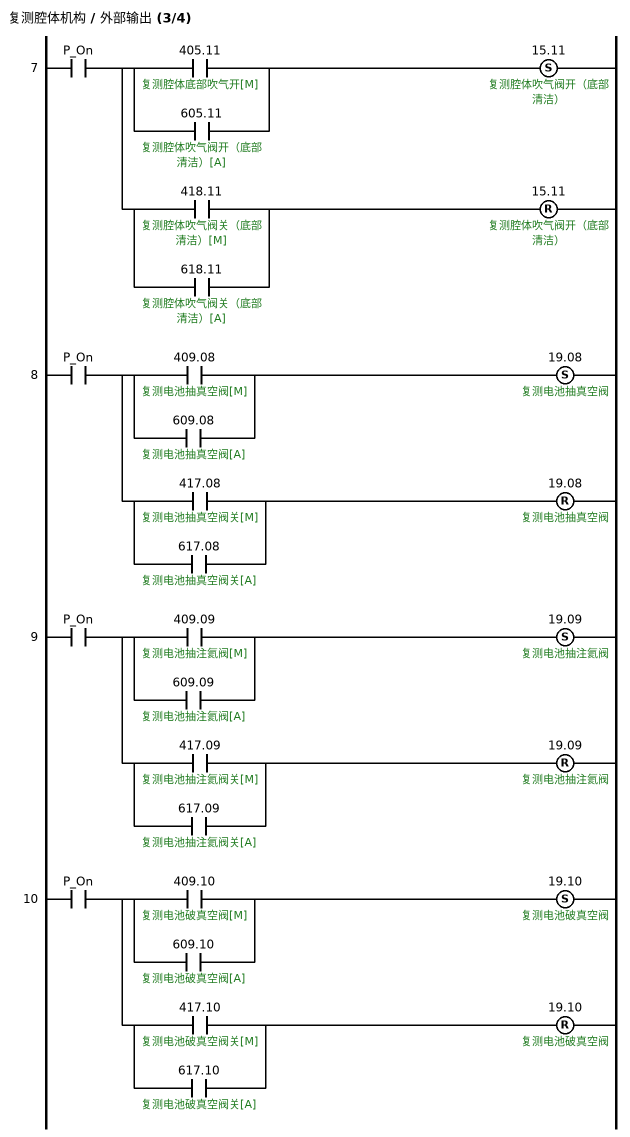
; [picture p624: 复测腔体机构 / 外部输出, rungs 7-10]
; rung 7
LD P_On
OUT TR0
LD 405.11  ; 复测腔体底部吹气开[M]
OR 605.11  ; 复测腔体吹气阀开（底部清洁）[A]
ANDLD
SET 15.11  ; 复测腔体吹气阀开（底部清洁）
LD TR0
LD 418.11  ; 复测腔体吹气阀关（底部清洁）[M]
OR 618.11  ; 复测腔体吹气阀关（底部清洁）[A]
ANDLD
RSET 15.11  ; 复测腔体吹气阀开（底部清洁）
; rung 8
LD P_On
OUT TR0
LD 409.08  ; 复测电池抽真空阀[M]
OR 609.08  ; 复测电池抽真空阀[A]
ANDLD
SET 19.08  ; 复测电池抽真空阀
LD TR0
LD 417.08  ; 复测电池抽真空阀关[M]
OR 617.08  ; 复测电池抽真空阀关[A]
ANDLD
RSET 19.08  ; 复测电池抽真空阀
; rung 9
LD P_On
OUT TR0
LD 409.09  ; 复测电池抽注氦阀[M]
OR 609.09  ; 复测电池抽注氦阀[A]
ANDLD
SET 19.09  ; 复测电池抽注氦阀
LD TR0
LD 417.09  ; 复测电池抽注氦阀关[M]
OR 617.09  ; 复测电池抽注氦阀关[A]
ANDLD
RSET 19.09  ; 复测电池抽注氦阀
; rung 10
LD P_On
OUT TR0
LD 409.10  ; 复测电池破真空阀[M]
OR 609.10  ; 复测电池破真空阀[A]
ANDLD
SET 19.10  ; 复测电池破真空阀
LD TR0
LD 417.10  ; 复测电池破真空阀关[M]
OR 617.10  ; 复测电池破真空阀关[A]
ANDLD
RSET 19.10  ; 复测电池破真空阀

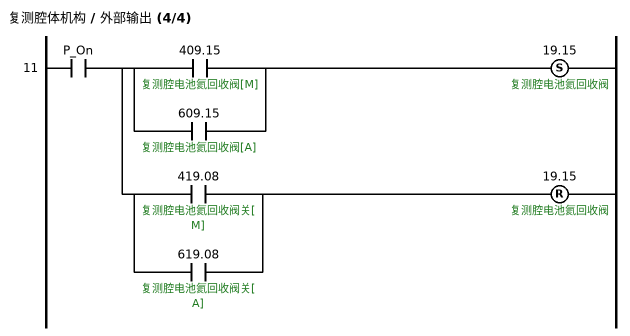
; rung 11
LD P_On
OUT TR0
LD 409.15  ; 复测腔电池氦回收阀[M]
OR 609.15  ; 复测腔电池氦回收阀[A]
ANDLD
SET 19.15  ; 复测腔电池氦回收阀
LD TR0
LD 419.08  ; 复测腔电池氦回收阀关[M]
OR 619.08  ; 复测腔电池氦回收阀关[A]
ANDLD
RSET 19.15  ; 复测腔电池氦回收阀

### Section END
; rung 0
END(001)

## Program Common (cyclic task 8)

### Section 动作延时

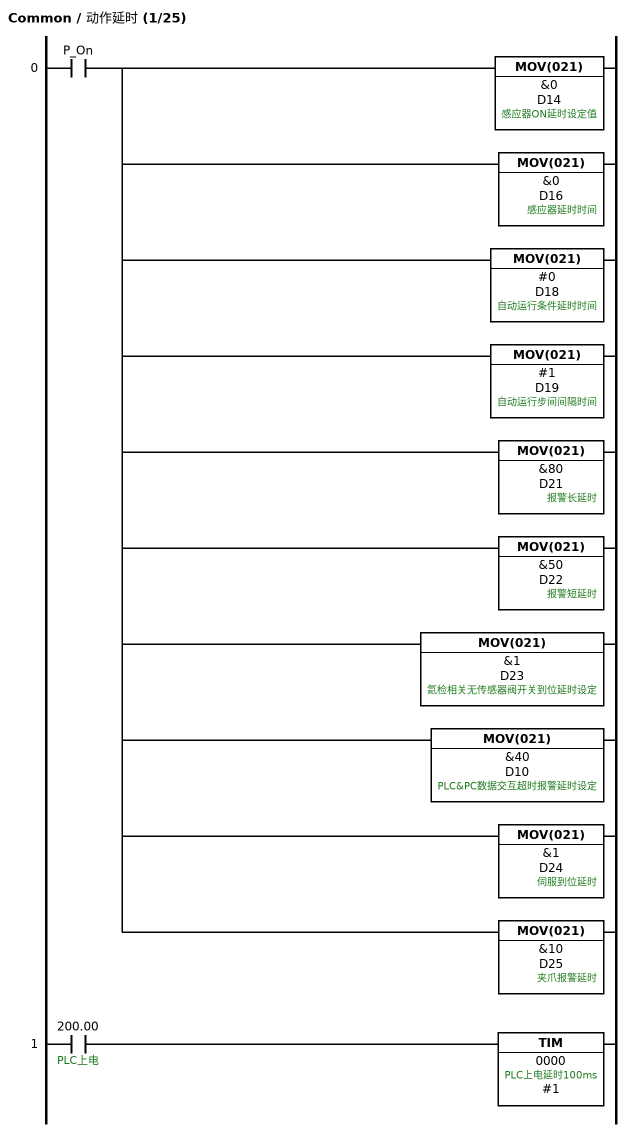
; rung 0
LD P_On
MOV(021) &0 D14  ; 感应器ON延时设定值
MOV(021) &0 D16  ; 感应器延时时间
MOV(021) #0 D18  ; 自动运行条件延时时间
MOV(021) #1 D19  ; 自动运行步间间隔时间
MOV(021) &80 D21  ; 报警长延时
MOV(021) &50 D22  ; 报警短延时
MOV(021) &1 D23  ; 氦检相关无传感器阀开关到位延时设定
MOV(021) &40 D10  ; PLC&PC数据交互超时报警延时设定
MOV(021) &1 D24  ; 伺服到位延时
MOV(021) &10 D25  ; 夹爪报警延时
; rung 1
LD 200.00  ; PLC上电
TIM 0000 #1  ; PLC上电延时100ms

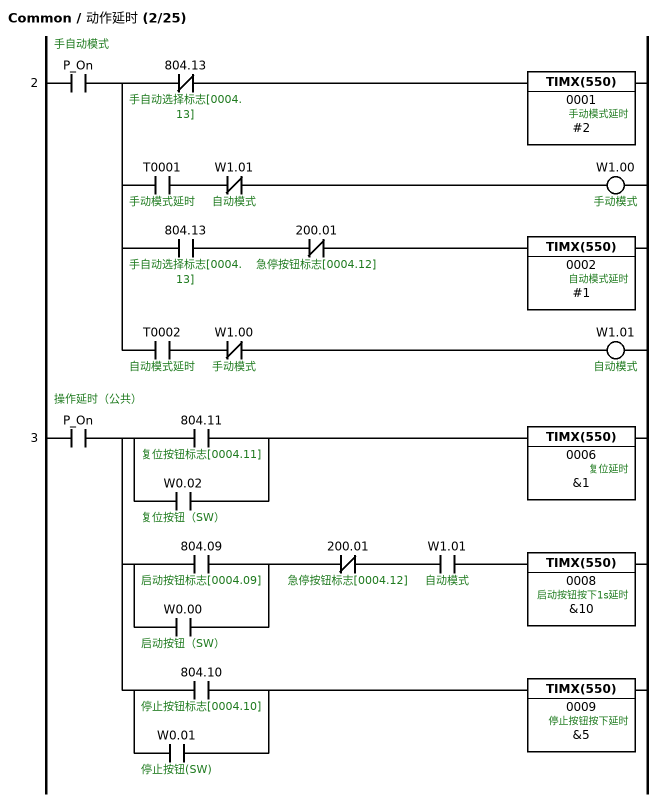
; rung 2: 手自动模式
LD P_On
OUT TR0
ANDNOT 804.13  ; 手自动选择标志[0004.13]
TIMX(550) 0001 #2  ; 手动模式延时
LD TR0
AND T0001  ; 手动模式延时
ANDNOT W1.01  ; 自动模式
OUT W1.00  ; 手动模式
LD TR0
AND 804.13  ; 手自动选择标志[0004.13]
ANDNOT 200.01  ; 急停按钮标志[0004.12]
TIMX(550) 0002 #1  ; 自动模式延时
LD TR0
AND T0002  ; 自动模式延时
ANDNOT W1.00  ; 手动模式
OUT W1.01  ; 自动模式
; rung 3: 操作延时（公共）
LD P_On
OUT TR0
LD 804.11  ; 复位按钮标志[0004.11]
OR W0.02  ; 复位按钮（SW）
ANDLD
TIMX(550) 0006 &1  ; 复位延时
LD TR0
LD 804.09  ; 启动按钮标志[0004.09]
OR W0.00  ; 启动按钮（SW）
ANDLD
ANDNOT 200.01  ; 急停按钮标志[0004.12]
AND W1.01  ; 自动模式
TIMX(550) 0008 &10  ; 启动按钮按下1s延时
LD TR0
LD 804.10  ; 停止按钮标志[0004.10]
OR W0.01  ; 停止按钮(SW)
ANDLD
TIMX(550) 0009 &5  ; 停止按钮按下延时

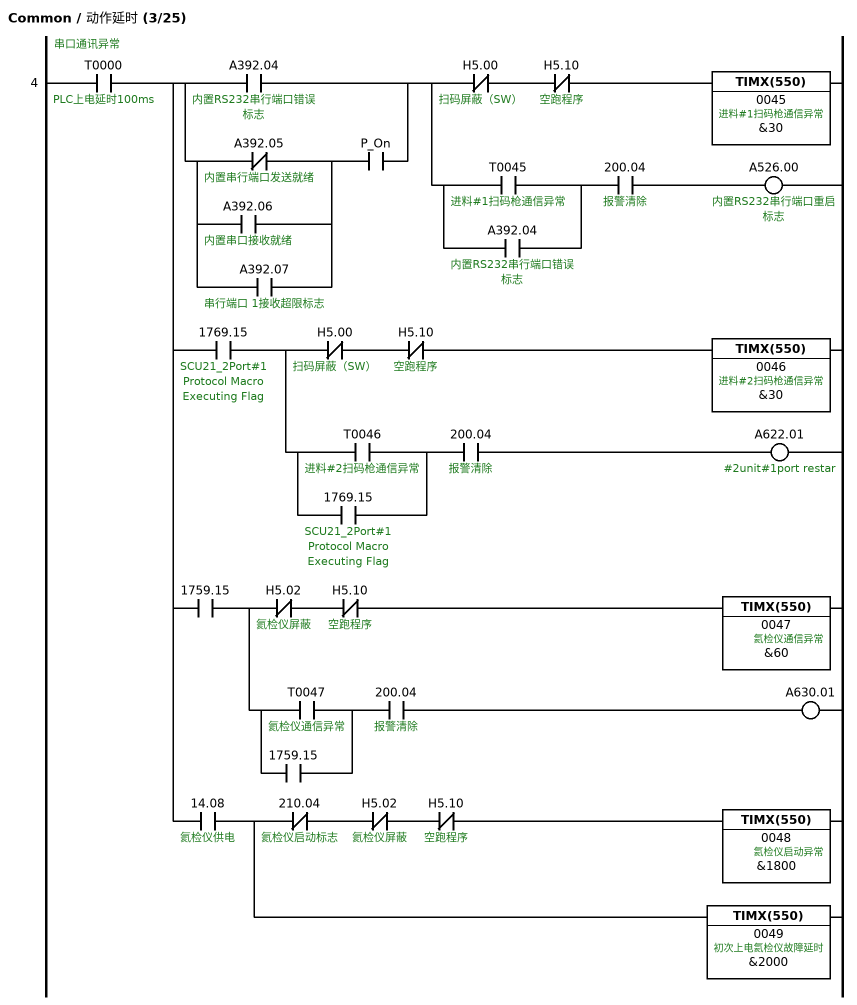
; rung 4: 串口通讯异常
LD T0000  ; PLC上电延时100ms
OUT TR0
LD A392.04  ; 内置RS232串行端口错误标志
LDNOT A392.05  ; 内置串行端口发送就绪
OR A392.06  ; 内置串口接收就绪
OR A392.07  ; 串行端口 1接收超限标志
AND P_On
ORLD
ANDLD
OUT TR1
ANDNOT H5.00  ; 扫码屏蔽（SW）
ANDNOT H5.10  ; 空跑程序
TIMX(550) 0045 &30  ; 进料#1扫码枪通信异常
LD TR1
LD T0045  ; 进料#1扫码枪通信异常
OR A392.04  ; 内置RS232串行端口错误标志
ANDLD
AND 200.04  ; 报警清除
OUT A526.00  ; 内置RS232串行端口重启标志
LD TR0
AND 1769.15  ; SCU21_2Port#1 Protocol Macro Executing Flag
OUT TR1
ANDNOT H5.00  ; 扫码屏蔽（SW）
ANDNOT H5.10  ; 空跑程序
TIMX(550) 0046 &30  ; 进料#2扫码枪通信异常
LD TR1
LD T0046  ; 进料#2扫码枪通信异常
OR 1769.15  ; SCU21_2Port#1 Protocol Macro Executing Flag
ANDLD
AND 200.04  ; 报警清除
OUT A622.01  ; #2unit#1port restar
LD TR0
AND 1759.15
OUT TR1
ANDNOT H5.02  ; 氦检仪屏蔽
ANDNOT H5.10  ; 空跑程序
TIMX(550) 0047 &60  ; 氦检仪通信异常
LD TR1
LD T0047  ; 氦检仪通信异常
OR 1759.15
ANDLD
AND 200.04  ; 报警清除
OUT A630.01
LD TR0
AND 14.08  ; 氦检仪供电
OUT TR0
ANDNOT 210.04  ; 氦检仪启动标志
ANDNOT H5.02  ; 氦检仪屏蔽
ANDNOT H5.10  ; 空跑程序
TIMX(550) 0048 &1800  ; 氦检仪启动异常
LD TR0
TIMX(550) 0049 &2000  ; 初次上电氦检仪故障延时

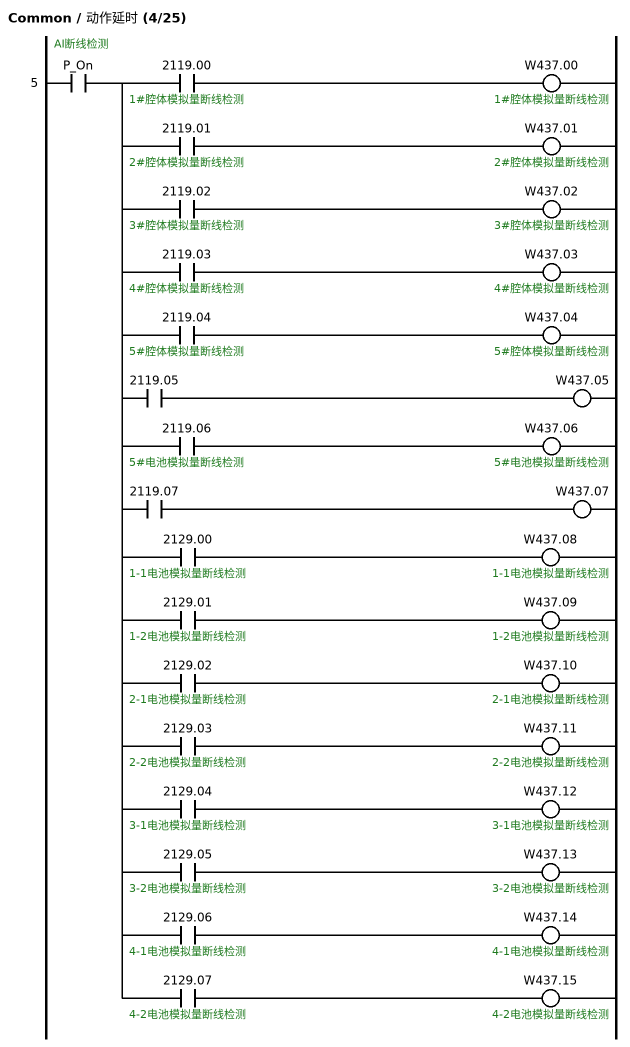
; rung 5: AI断线检测
LD P_On
OUT TR0
AND 2119.00  ; 1#腔体模拟量断线检测
OUT W437.00  ; 1#腔体模拟量断线检测
LD TR0
AND 2119.01  ; 2#腔体模拟量断线检测
OUT W437.01  ; 2#腔体模拟量断线检测
LD TR0
AND 2119.02  ; 3#腔体模拟量断线检测
OUT W437.02  ; 3#腔体模拟量断线检测
LD TR0
AND 2119.03  ; 4#腔体模拟量断线检测
OUT W437.03  ; 4#腔体模拟量断线检测
LD TR0
AND 2119.04  ; 5#腔体模拟量断线检测
OUT W437.04  ; 5#腔体模拟量断线检测
LD TR0
AND 2119.05
OUT W437.05
LD TR0
AND 2119.06  ; 5#电池模拟量断线检测
OUT W437.06  ; 5#电池模拟量断线检测
LD TR0
AND 2119.07
OUT W437.07
LD TR0
AND 2129.00  ; 1-1电池模拟量断线检测
OUT W437.08  ; 1-1电池模拟量断线检测
LD TR0
AND 2129.01  ; 1-2电池模拟量断线检测
OUT W437.09  ; 1-2电池模拟量断线检测
LD TR0
AND 2129.02  ; 2-1电池模拟量断线检测
OUT W437.10  ; 2-1电池模拟量断线检测
LD TR0
AND 2129.03  ; 2-2电池模拟量断线检测
OUT W437.11  ; 2-2电池模拟量断线检测
LD TR0
AND 2129.04  ; 3-1电池模拟量断线检测
OUT W437.12  ; 3-1电池模拟量断线检测
LD TR0
AND 2129.05  ; 3-2电池模拟量断线检测
OUT W437.13  ; 3-2电池模拟量断线检测
LD TR0
AND 2129.06  ; 4-1电池模拟量断线检测
OUT W437.14  ; 4-1电池模拟量断线检测
LD TR0
AND 2129.07  ; 4-2电池模拟量断线检测
OUT W437.15  ; 4-2电池模拟量断线检测

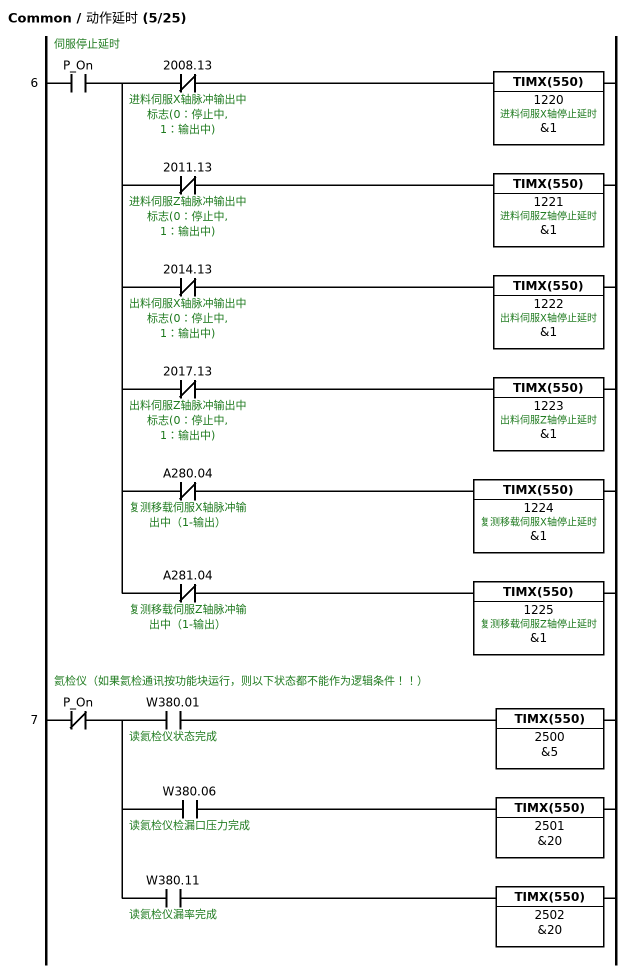
; rung 6: 伺服停止延时
LD P_On
OUT TR0
ANDNOT 2008.13  ; 进料伺服X轴脉冲输出中标志(0：停止中,1：输出中)
TIMX(550) 1220 &1  ; 进料伺服X轴停止延时
LD TR0
ANDNOT 2011.13  ; 进料伺服Z轴脉冲输出中标志(0：停止中,1：输出中)
TIMX(550) 1221 &1  ; 进料伺服Z轴停止延时
LD TR0
ANDNOT 2014.13  ; 出料伺服X轴脉冲输出中标志(0：停止中,1：输出中)
TIMX(550) 1222 &1  ; 出料伺服X轴停止延时
LD TR0
ANDNOT 2017.13  ; 出料伺服Z轴脉冲输出中标志(0：停止中,1：输出中)
TIMX(550) 1223 &1  ; 出料伺服Z轴停止延时
LD TR0
ANDNOT A280.04  ; 复测移载伺服X轴脉冲输出中（1-输出）
TIMX(550) 1224 &1  ; 复测移载伺服X轴停止延时
LD TR0
ANDNOT A281.04  ; 复测移载伺服Z轴脉冲输出中（1-输出）
TIMX(550) 1225 &1  ; 复测移载伺服Z轴停止延时
; rung 7: 氦检仪（如果氦检通讯按功能块运行，则以下状态都不能作为逻辑条件！！）
LDNOT P_On
OUT TR0
AND W380.01  ; 读氦检仪状态完成
TIMX(550) 2500 &5
LD TR0
AND W380.06  ; 读氦检仪检漏口压力完成
TIMX(550) 2501 &20
LD TR0
AND W380.11  ; 读氦检仪漏率完成
TIMX(550) 2502 &20

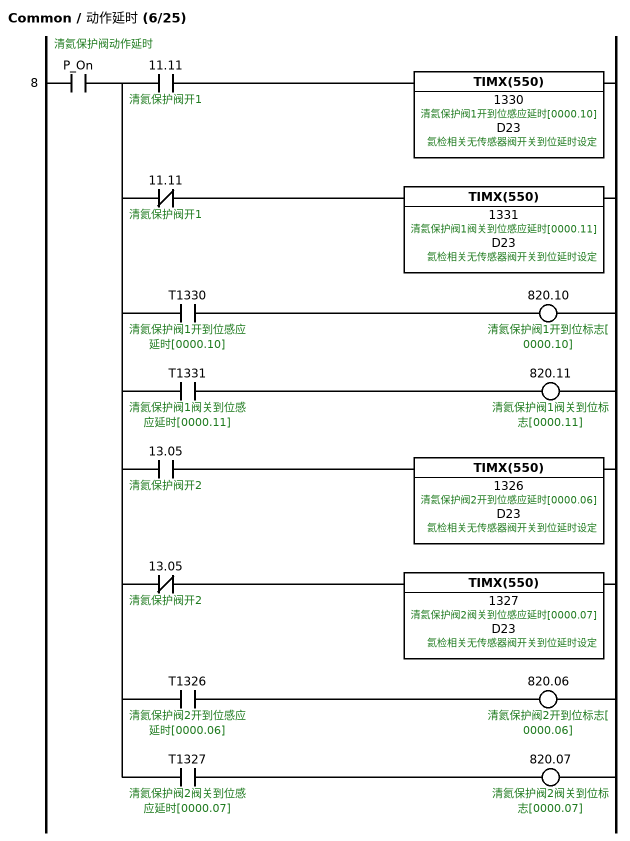
; rung 8: 清氦保护阀动作延时
LD P_On
OUT TR0
AND 11.11  ; 清氦保护阀开1
TIMX(550) 1330 D23  ; 氦检相关无传感器阀开关到位延时设定, 清氦保护阀1开到位感应延时[0000.10]
LD TR0
ANDNOT 11.11  ; 清氦保护阀开1
TIMX(550) 1331 D23  ; 氦检相关无传感器阀开关到位延时设定, 清氦保护阀1阀关到位感应延时[0000.11]
LD TR0
AND T1330  ; 清氦保护阀1开到位感应延时[0000.10]
OUT 820.10  ; 清氦保护阀1开到位标志[0000.10]
LD TR0
AND T1331  ; 清氦保护阀1阀关到位感应延时[0000.11]
OUT 820.11  ; 清氦保护阀1阀关到位标志[0000.11]
LD TR0
AND 13.05  ; 清氦保护阀开2
TIMX(550) 1326 D23  ; 氦检相关无传感器阀开关到位延时设定, 清氦保护阀2开到位感应延时[0000.06]
LD TR0
ANDNOT 13.05  ; 清氦保护阀开2
TIMX(550) 1327 D23  ; 氦检相关无传感器阀开关到位延时设定, 清氦保护阀2阀关到位感应延时[0000.07]
LD TR0
AND T1326  ; 清氦保护阀2开到位感应延时[0000.06]
OUT 820.06  ; 清氦保护阀2开到位标志[0000.06]
LD TR0
AND T1327  ; 清氦保护阀2阀关到位感应延时[0000.07]
OUT 820.07  ; 清氦保护阀2阀关到位标志[0000.07]

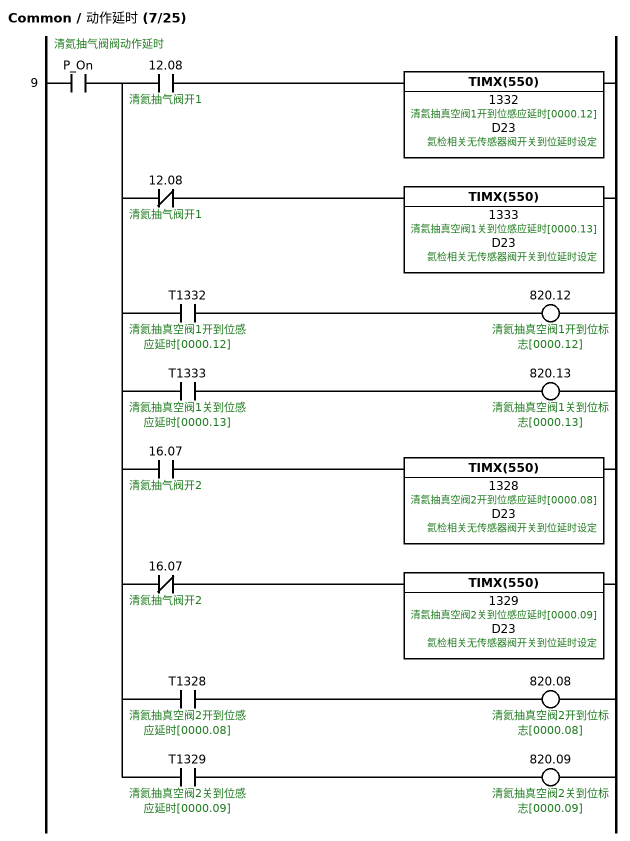
; rung 9: 清氦抽气阀阀动作延时
LD P_On
OUT TR0
AND 12.08  ; 清氦抽气阀开1
TIMX(550) 1332 D23  ; 氦检相关无传感器阀开关到位延时设定, 清氦抽真空阀1开到位感应延时[0000.12]
LD TR0
ANDNOT 12.08  ; 清氦抽气阀开1
TIMX(550) 1333 D23  ; 氦检相关无传感器阀开关到位延时设定, 清氦抽真空阀1关到位感应延时[0000.13]
LD TR0
AND T1332  ; 清氦抽真空阀1开到位感应延时[0000.12]
OUT 820.12  ; 清氦抽真空阀1开到位标志[0000.12]
LD TR0
AND T1333  ; 清氦抽真空阀1关到位感应延时[0000.13]
OUT 820.13  ; 清氦抽真空阀1关到位标志[0000.13]
LD TR0
AND 16.07  ; 清氦抽气阀开2
TIMX(550) 1328 D23  ; 氦检相关无传感器阀开关到位延时设定, 清氦抽真空阀2开到位感应延时[0000.08]
LD TR0
ANDNOT 16.07  ; 清氦抽气阀开2
TIMX(550) 1329 D23  ; 氦检相关无传感器阀开关到位延时设定, 清氦抽真空阀2关到位感应延时[0000.09]
LD TR0
AND T1328  ; 清氦抽真空阀2开到位感应延时[0000.08]
OUT 820.08  ; 清氦抽真空阀2开到位标志[0000.08]
LD TR0
AND T1329  ; 清氦抽真空阀2关到位感应延时[0000.09]
OUT 820.09  ; 清氦抽真空阀2关到位标志[0000.09]

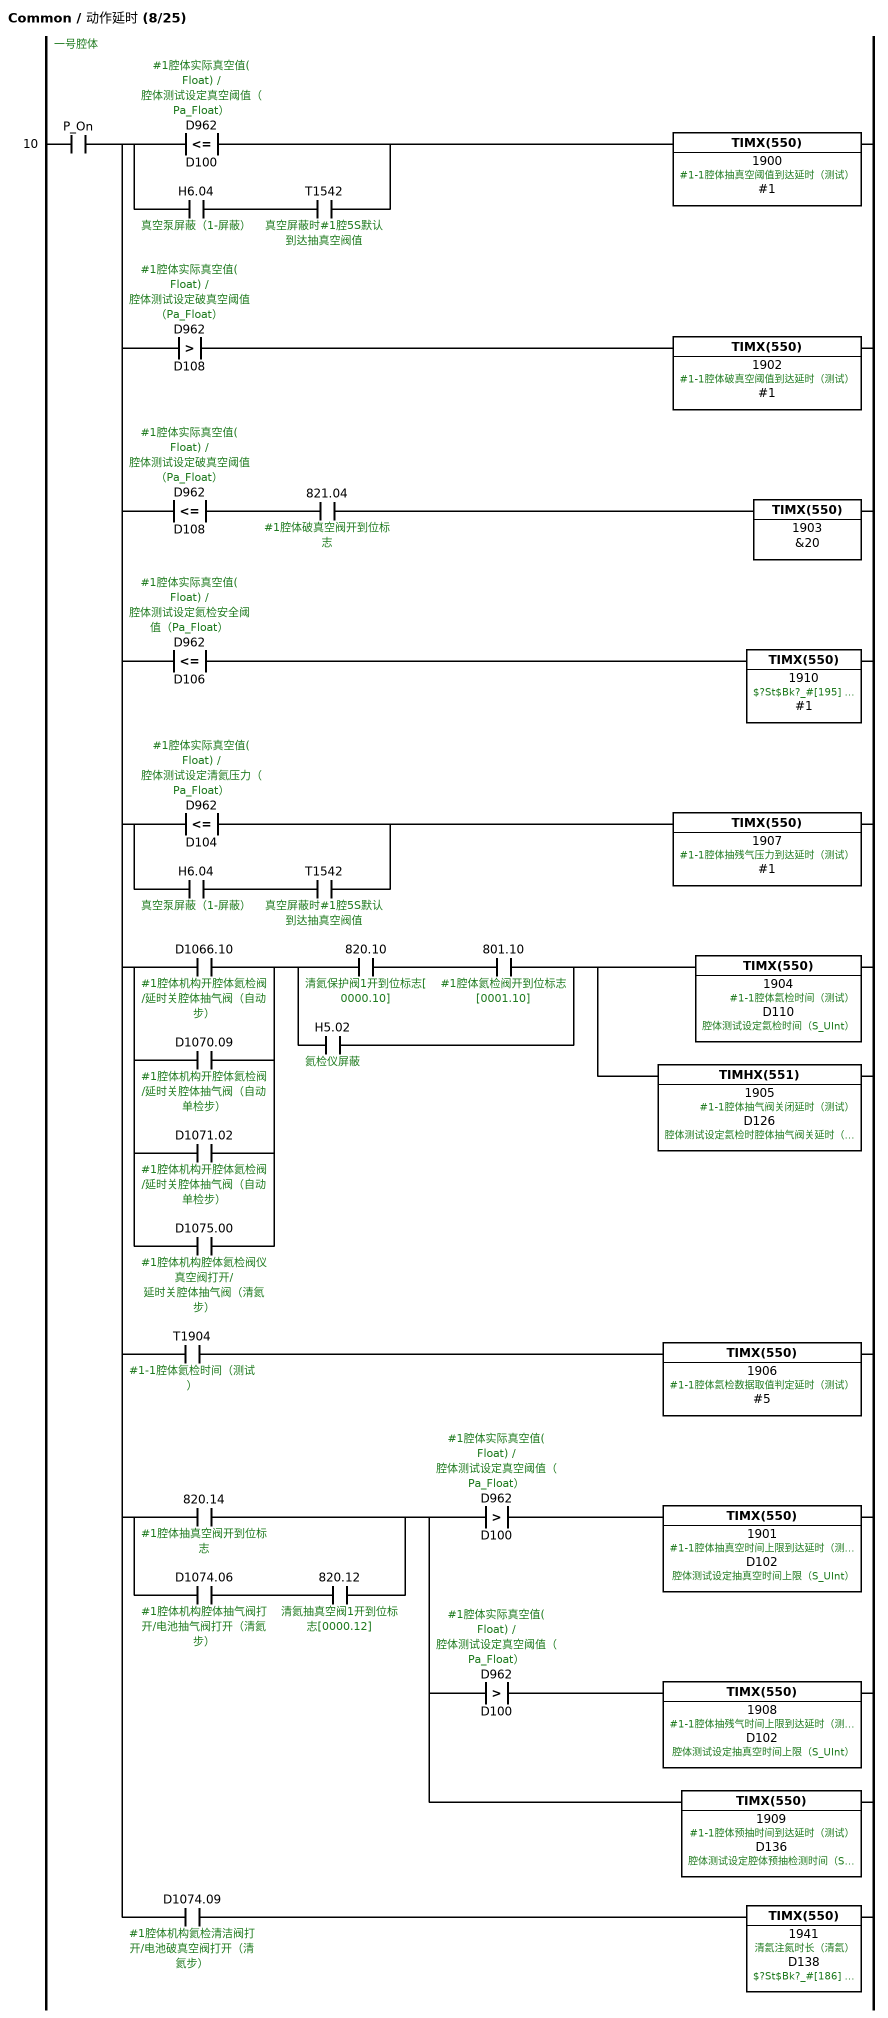
; rung 10: 一号腔体
LD P_On
OUT TR0
LD<=F(332) D962 D100  ; #1腔体实际真空值(Float), 腔体测试设定真空阈值（Pa_Float）
LD H6.04  ; 真空泵屏蔽（1-屏蔽）
AND T1542  ; 真空屏蔽时#1腔5S默认到达抽真空阀值
ORLD
ANDLD
TIMX(550) 1900 #1  ; #1-1腔体抽真空阈值到达延时（测试）
LD TR0
AND>F(333) D962 D108  ; #1腔体实际真空值(Float), 腔体测试设定破真空阈值（Pa_Float）
TIMX(550) 1902 #1  ; #1-1腔体破真空阈值到达延时（测试）
LD TR0
AND<=F(332) D962 D108  ; #1腔体实际真空值(Float), 腔体测试设定破真空阈值（Pa_Float）
AND 821.04  ; #1腔体破真空阀开到位标志
TIMX(550) 1903 &20
LD TR0
AND<=F(332) D962 D106  ; #1腔体实际真空值(Float), 腔体测试设定氦检安全阈值（Pa_Float）
TIMX(550) 1910 #1  ; $?St$Bk?_#[195] / #1-1腔体真空在可氦检状态（测试） / $?St$Bk?_#[195]
LD TR0
LD<=F(332) D962 D104  ; #1腔体实际真空值(Float), 腔体测试设定清氦压力（Pa_Float）
LD H6.04  ; 真空泵屏蔽（1-屏蔽）
AND T1542  ; 真空屏蔽时#1腔5S默认到达抽真空阀值
ORLD
ANDLD
TIMX(550) 1907 #1  ; #1-1腔体抽残气压力到达延时（测试）
LD TR0
LD D1066.10  ; #1腔体机构开腔体氦检阀/延时关腔体抽气阀（自动步）
OR D1070.09  ; #1腔体机构开腔体氦检阀/延时关腔体抽气阀（自动单检步）
OR D1071.02  ; #1腔体机构开腔体氦检阀/延时关腔体抽气阀（自动单检步）
OR D1075.00  ; #1腔体机构腔体氦检阀仪真空阀打开/延时关腔体抽气阀（清氦步）
ANDLD
LD 820.10  ; 清氦保护阀1开到位标志[0000.10]
AND 801.10  ; #1腔体氦检阀开到位标志[0001.10]
OR H5.02  ; 氦检仪屏蔽
ANDLD
TIMX(550) 1904 D110  ; 腔体测试设定氦检时间（S_UInt）, #1-1腔体氦检时间（测试）
TIMHX(551) 1905 D126  ; 腔体测试设定氦检时腔体抽气阀关延时（S_UInt）, #1-1腔体抽气阀关闭延时（测试）
LD TR0
AND T1904  ; #1-1腔体氦检时间（测试）
TIMX(550) 1906 #5  ; #1-1腔体氦检数据取值判定延时（测试）
LD TR0
LD 820.14  ; #1腔体抽真空阀开到位标志
LD D1074.06  ; #1腔体机构腔体抽气阀打开/电池抽气阀打开（清氦步）
AND 820.12  ; 清氦抽真空阀1开到位标志[0000.12]
ORLD
ANDLD
OUT TR1
AND>F(333) D962 D100  ; #1腔体实际真空值(Float), 腔体测试设定真空阈值（Pa_Float）
TIMX(550) 1901 D102  ; 腔体测试设定抽真空时间上限（S_UInt）, #1-1腔体抽真空时间上限到达延时（测试）
LD TR1
AND>F(333) D962 D100  ; #1腔体实际真空值(Float), 腔体测试设定真空阈值（Pa_Float）
TIMX(550) 1908 D102  ; 腔体测试设定抽真空时间上限（S_UInt）, #1-1腔体抽残气时间上限到达延时（测试）
LD TR1
TIMX(550) 1909 D136  ; 腔体测试设定腔体预抽检测时间（S_UInt）, #1-1腔体预抽时间到达延时（测试）
LD TR0
AND D1074.09  ; #1腔体机构氦检清洁阀打开/电池破真空阀打开（清氦步）
TIMX(550) 1941 D138  ; $?St$Bk?_#[186] / 管路清氦注氮时间（S_UInt） / $?St$Bk?_#[186], 清氦注氮时长（清氦）

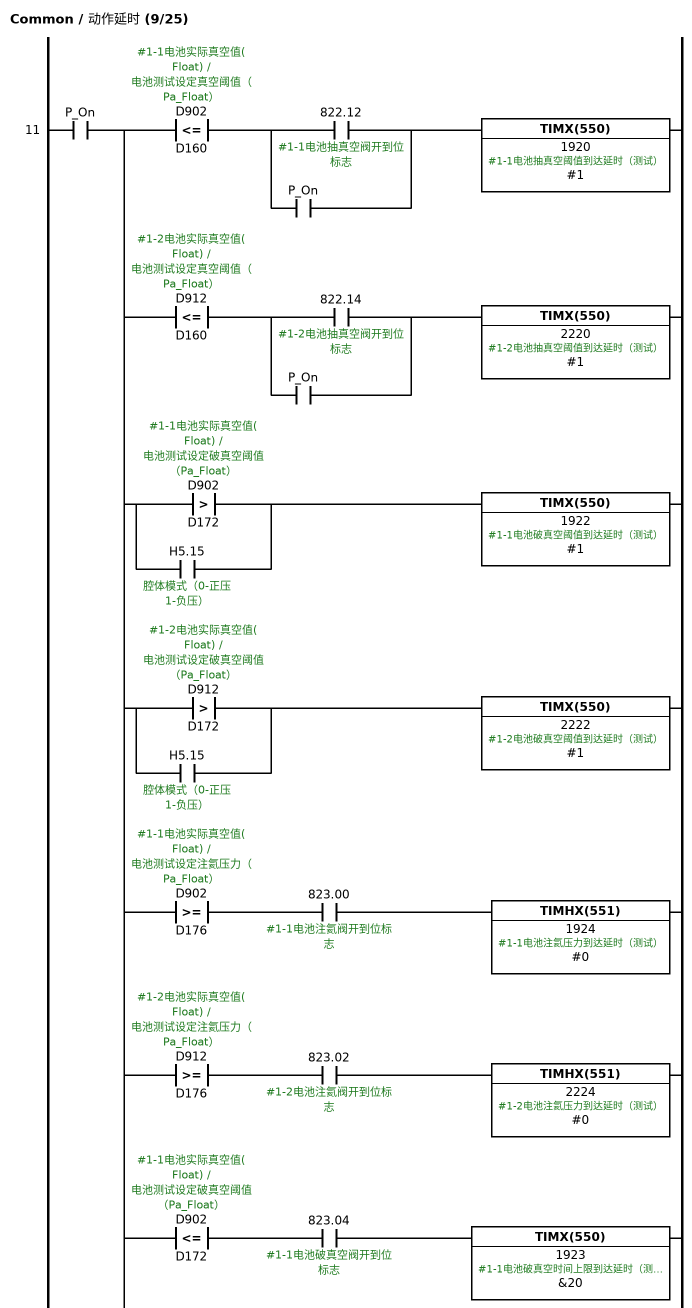

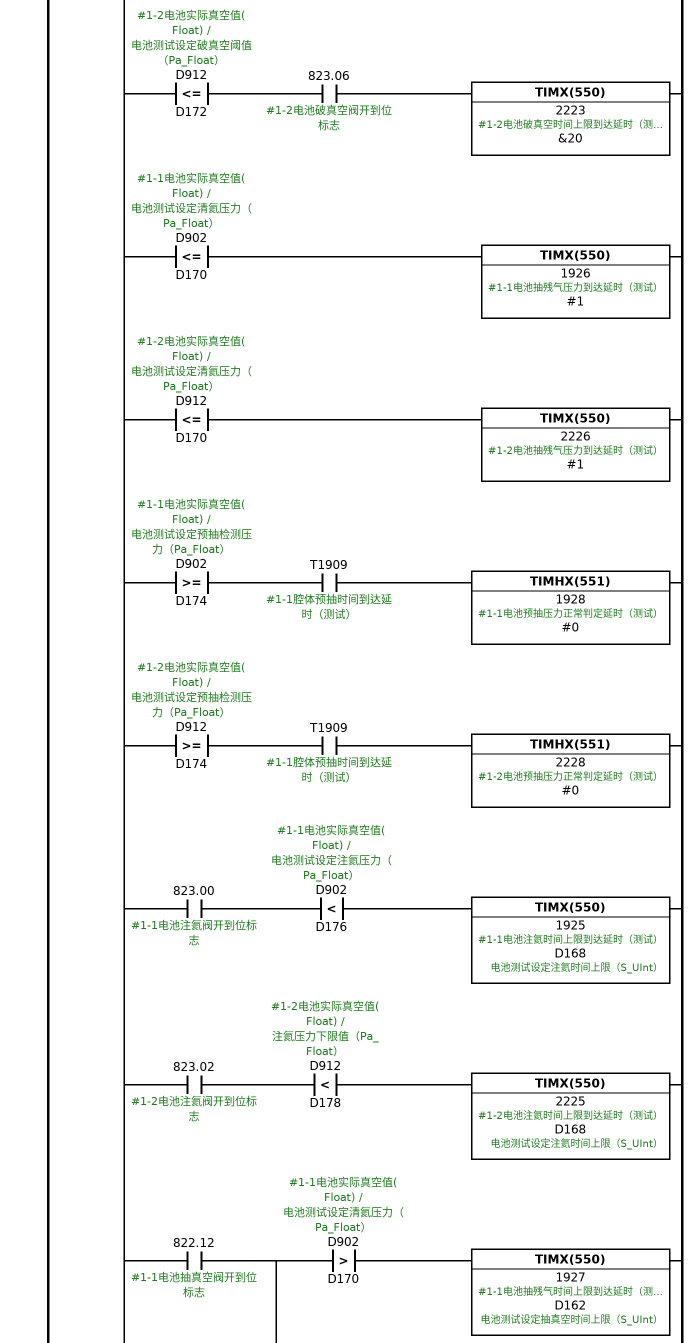

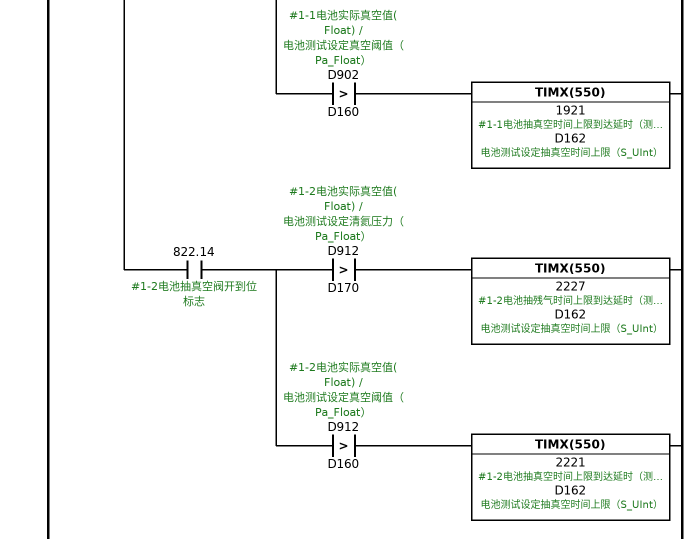
; rung 11
LD P_On
OUT TR0
AND<=F(332) D902 D160  ; #1-1电池实际真空值(Float), 电池测试设定真空阈值（Pa_Float）
LD 822.12  ; #1-1电池抽真空阀开到位标志
OR P_On
ANDLD
TIMX(550) 1920 #1  ; #1-1电池抽真空阈值到达延时（测试）
LD TR0
AND<=F(332) D912 D160  ; #1-2电池实际真空值(Float), 电池测试设定真空阈值（Pa_Float）
LD 822.14  ; #1-2电池抽真空阀开到位标志
OR P_On
ANDLD
TIMX(550) 2220 #1  ; #1-2电池抽真空阈值到达延时（测试）
LD TR0
LD>F(333) D902 D172  ; #1-1电池实际真空值(Float), 电池测试设定破真空阈值（Pa_Float）
OR H5.15  ; 腔体模式（0-正压 1-负压）
ANDLD
TIMX(550) 1922 #1  ; #1-1电池破真空阈值到达延时（测试）
LD TR0
LD>F(333) D912 D172  ; #1-2电池实际真空值(Float), 电池测试设定破真空阈值（Pa_Float）
OR H5.15  ; 腔体模式（0-正压 1-负压）
ANDLD
TIMX(550) 2222 #1  ; #1-2电池破真空阈值到达延时（测试）
LD TR0
AND>=F(334) D902 D176  ; #1-1电池实际真空值(Float), 电池测试设定注氦压力（Pa_Float）
AND 823.00  ; #1-1电池注氦阀开到位标志
TIMHX(551) 1924 #0  ; #1-1电池注氦压力到达延时（测试）
LD TR0
AND>=F(334) D912 D176  ; #1-2电池实际真空值(Float), 电池测试设定注氦压力（Pa_Float）
AND 823.02  ; #1-2电池注氦阀开到位标志
TIMHX(551) 2224 #0  ; #1-2电池注氦压力到达延时（测试）
LD TR0
AND<=F(332) D902 D172  ; #1-1电池实际真空值(Float), 电池测试设定破真空阈值（Pa_Float）
AND 823.04  ; #1-1电池破真空阀开到位标志
TIMX(550) 1923 &20  ; #1-1电池破真空时间上限到达延时（测试）
LD TR0
AND<=F(332) D912 D172  ; #1-2电池实际真空值(Float), 电池测试设定破真空阈值（Pa_Float）
AND 823.06  ; #1-2电池破真空阀开到位标志
TIMX(550) 2223 &20  ; #1-2电池破真空时间上限到达延时（测试）
LD TR0
AND<=F(332) D902 D170  ; #1-1电池实际真空值(Float), 电池测试设定清氦压力（Pa_Float）
TIMX(550) 1926 #1  ; #1-1电池抽残气压力到达延时（测试）
LD TR0
AND<=F(332) D912 D170  ; #1-2电池实际真空值(Float), 电池测试设定清氦压力（Pa_Float）
TIMX(550) 2226 #1  ; #1-2电池抽残气压力到达延时（测试）
LD TR0
AND>=F(334) D902 D174  ; #1-1电池实际真空值(Float), 电池测试设定预抽检测压力（Pa_Float）
AND T1909  ; #1-1腔体预抽时间到达延时（测试）
TIMHX(551) 1928 #0  ; #1-1电池预抽压力正常判定延时（测试）
LD TR0
AND>=F(334) D912 D174  ; #1-2电池实际真空值(Float), 电池测试设定预抽检测压力（Pa_Float）
AND T1909  ; #1-1腔体预抽时间到达延时（测试）
TIMHX(551) 2228 #0  ; #1-2电池预抽压力正常判定延时（测试）
LD TR0
AND 823.00  ; #1-1电池注氦阀开到位标志
AND<F(331) D902 D176  ; #1-1电池实际真空值(Float), 电池测试设定注氦压力（Pa_Float）
TIMX(550) 1925 D168  ; 电池测试设定注氦时间上限（S_UInt）, #1-1电池注氦时间上限到达延时（测试）
LD TR0
AND 823.02  ; #1-2电池注氦阀开到位标志
AND<F(331) D912 D178  ; #1-2电池实际真空值(Float), 注氦压力下限值（Pa_Float）
TIMX(550) 2225 D168  ; 电池测试设定注氦时间上限（S_UInt）, #1-2电池注氦时间上限到达延时（测试）
LD TR0
AND 822.12  ; #1-1电池抽真空阀开到位标志
OUT TR1
AND>F(333) D902 D170  ; #1-1电池实际真空值(Float), 电池测试设定清氦压力（Pa_Float）
TIMX(550) 1927 D162  ; 电池测试设定抽真空时间上限（S_UInt）, #1-1电池抽残气时间上限到达延时（测试）
LD TR1
AND>F(333) D902 D160  ; #1-1电池实际真空值(Float), 电池测试设定真空阈值（Pa_Float）
TIMX(550) 1921 D162  ; 电池测试设定抽真空时间上限（S_UInt）, #1-1电池抽真空时间上限到达延时（测试）
LD TR0
AND 822.14  ; #1-2电池抽真空阀开到位标志
OUT TR0
AND>F(333) D912 D170  ; #1-2电池实际真空值(Float), 电池测试设定清氦压力（Pa_Float）
TIMX(550) 2227 D162  ; 电池测试设定抽真空时间上限（S_UInt）, #1-2电池抽残气时间上限到达延时（测试）
LD TR0
AND>F(333) D912 D160  ; #1-2电池实际真空值(Float), 电池测试设定真空阈值（Pa_Float）
TIMX(550) 2221 D162  ; 电池测试设定抽真空时间上限（S_UInt）, #1-2电池抽真空时间上限到达延时（测试）

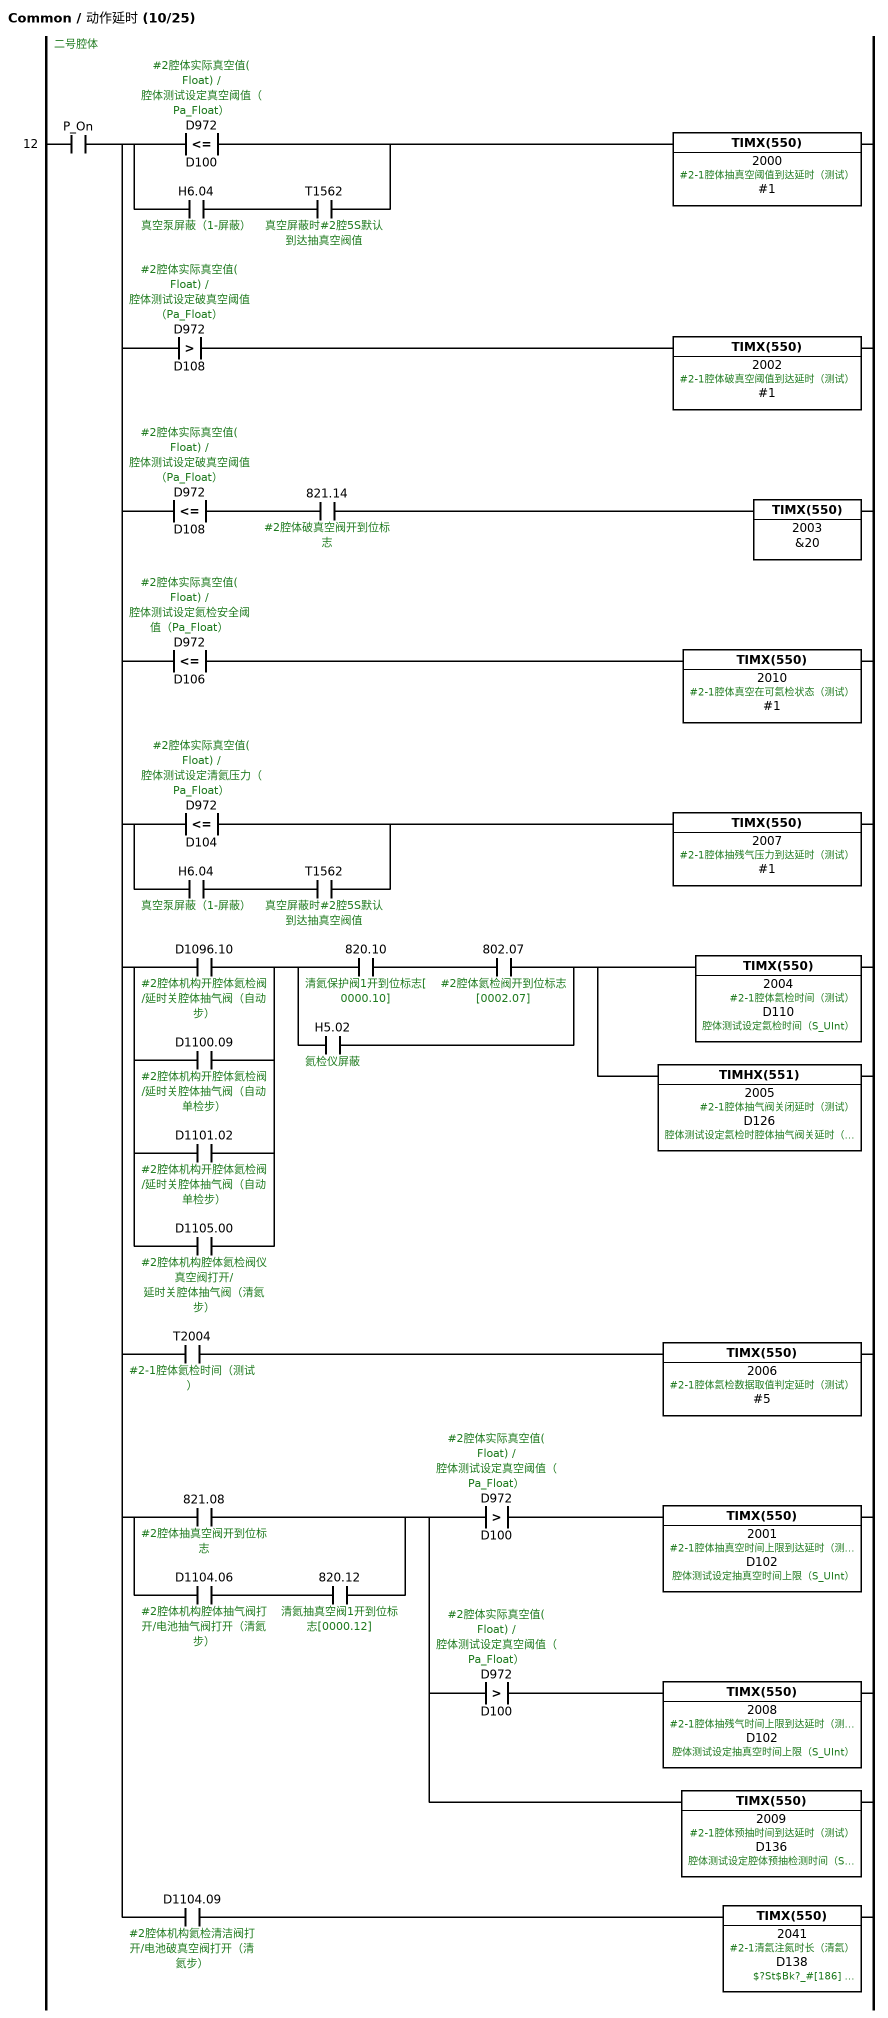
; rung 12: 二号腔体
LD P_On
OUT TR0
LD<=F(332) D972 D100  ; #2腔体实际真空值(Float), 腔体测试设定真空阈值（Pa_Float）
LD H6.04  ; 真空泵屏蔽（1-屏蔽）
AND T1562  ; 真空屏蔽时#2腔5S默认到达抽真空阀值
ORLD
ANDLD
TIMX(550) 2000 #1  ; #2-1腔体抽真空阈值到达延时（测试）
LD TR0
AND>F(333) D972 D108  ; #2腔体实际真空值(Float), 腔体测试设定破真空阈值（Pa_Float）
TIMX(550) 2002 #1  ; #2-1腔体破真空阈值到达延时（测试）
LD TR0
AND<=F(332) D972 D108  ; #2腔体实际真空值(Float), 腔体测试设定破真空阈值（Pa_Float）
AND 821.14  ; #2腔体破真空阀开到位标志
TIMX(550) 2003 &20
LD TR0
AND<=F(332) D972 D106  ; #2腔体实际真空值(Float), 腔体测试设定氦检安全阈值（Pa_Float）
TIMX(550) 2010 #1  ; #2-1腔体真空在可氦检状态（测试）
LD TR0
LD<=F(332) D972 D104  ; #2腔体实际真空值(Float), 腔体测试设定清氦压力（Pa_Float）
LD H6.04  ; 真空泵屏蔽（1-屏蔽）
AND T1562  ; 真空屏蔽时#2腔5S默认到达抽真空阀值
ORLD
ANDLD
TIMX(550) 2007 #1  ; #2-1腔体抽残气压力到达延时（测试）
LD TR0
LD D1096.10  ; #2腔体机构开腔体氦检阀/延时关腔体抽气阀（自动步）
OR D1100.09  ; #2腔体机构开腔体氦检阀/延时关腔体抽气阀（自动单检步）
OR D1101.02  ; #2腔体机构开腔体氦检阀/延时关腔体抽气阀（自动单检步）
OR D1105.00  ; #2腔体机构腔体氦检阀仪真空阀打开/延时关腔体抽气阀（清氦步）
ANDLD
LD 820.10  ; 清氦保护阀1开到位标志[0000.10]
AND 802.07  ; #2腔体氦检阀开到位标志[0002.07]
OR H5.02  ; 氦检仪屏蔽
ANDLD
TIMX(550) 2004 D110  ; 腔体测试设定氦检时间（S_UInt）, #2-1腔体氦检时间（测试）
TIMHX(551) 2005 D126  ; 腔体测试设定氦检时腔体抽气阀关延时（S_UInt）, #2-1腔体抽气阀关闭延时（测试）
LD TR0
AND T2004  ; #2-1腔体氦检时间（测试）
TIMX(550) 2006 #5  ; #2-1腔体氦检数据取值判定延时（测试）
LD TR0
LD 821.08  ; #2腔体抽真空阀开到位标志
LD D1104.06  ; #2腔体机构腔体抽气阀打开/电池抽气阀打开（清氦步）
AND 820.12  ; 清氦抽真空阀1开到位标志[0000.12]
ORLD
ANDLD
OUT TR1
AND>F(333) D972 D100  ; #2腔体实际真空值(Float), 腔体测试设定真空阈值（Pa_Float）
TIMX(550) 2001 D102  ; 腔体测试设定抽真空时间上限（S_UInt）, #2-1腔体抽真空时间上限到达延时（测试）
LD TR1
AND>F(333) D972 D100  ; #2腔体实际真空值(Float), 腔体测试设定真空阈值（Pa_Float）
TIMX(550) 2008 D102  ; 腔体测试设定抽真空时间上限（S_UInt）, #2-1腔体抽残气时间上限到达延时（测试）
LD TR1
TIMX(550) 2009 D136  ; 腔体测试设定腔体预抽检测时间（S_UInt）, #2-1腔体预抽时间到达延时（测试）
LD TR0
AND D1104.09  ; #2腔体机构氦检清洁阀打开/电池破真空阀打开（清氦步）
TIMX(550) 2041 D138  ; $?St$Bk?_#[186] / 管路清氦注氮时间（S_UInt） / $?St$Bk?_#[186], #2-1清氦注氮时长（清氦）

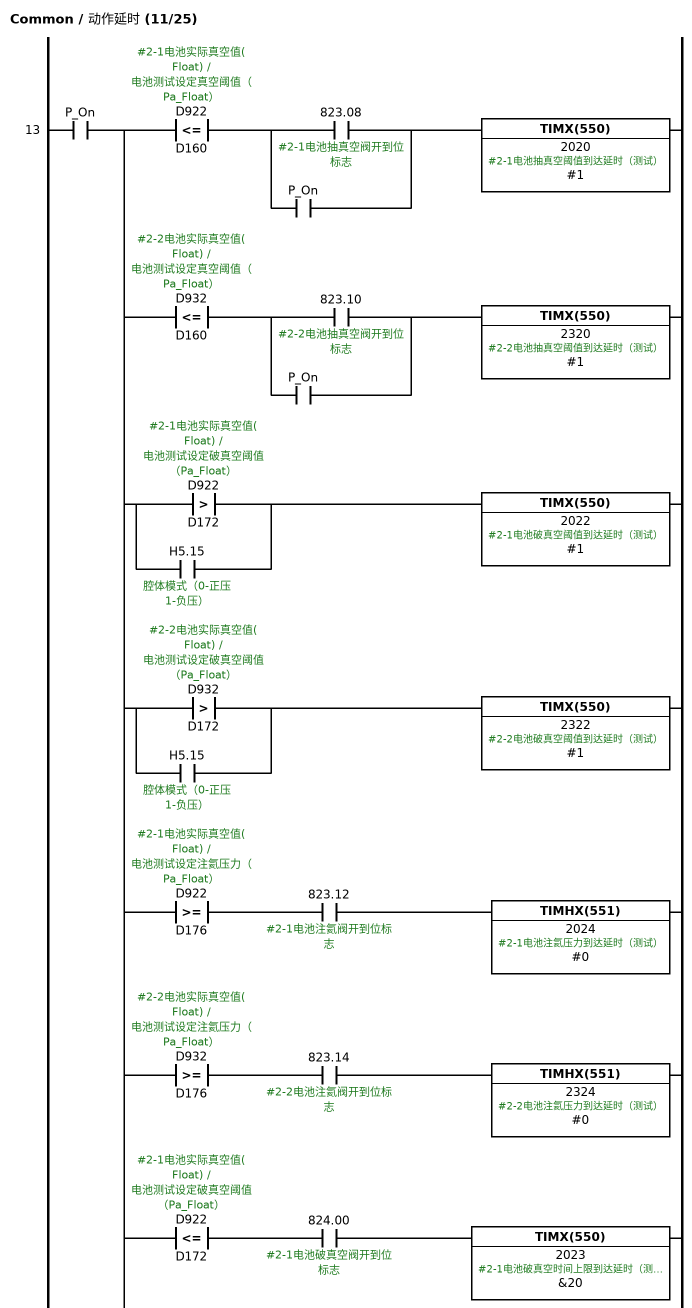

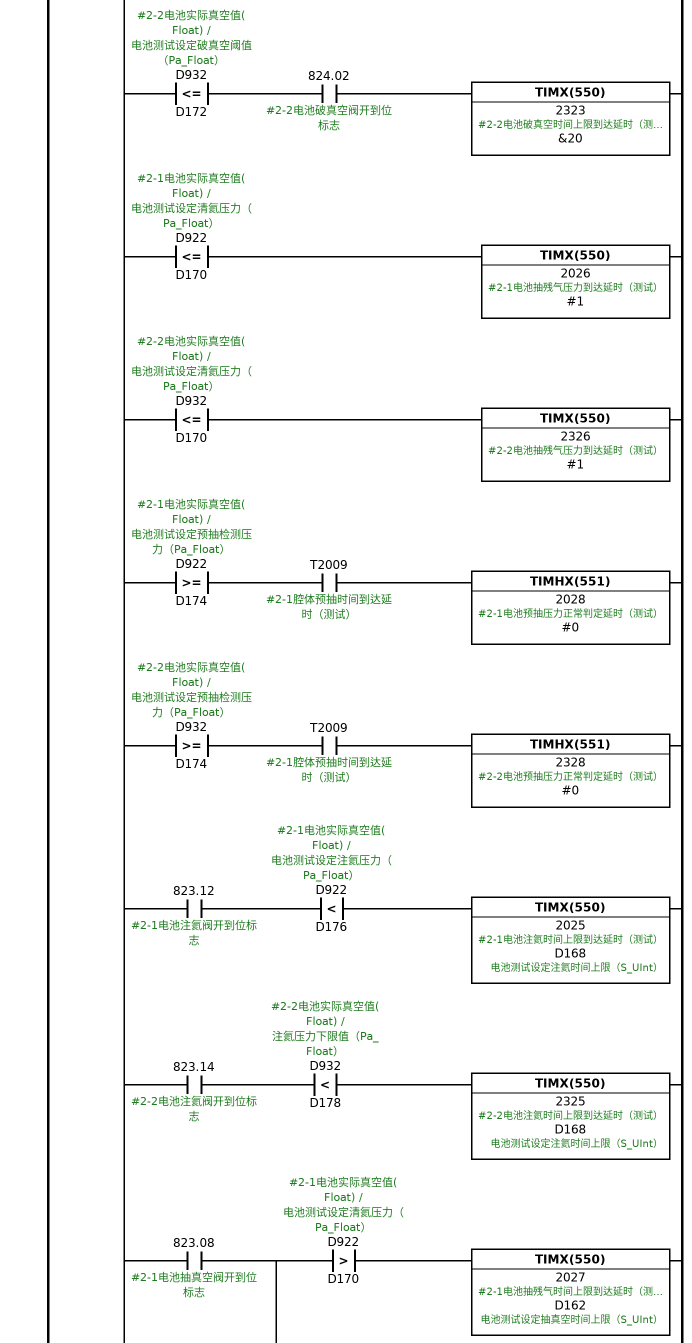

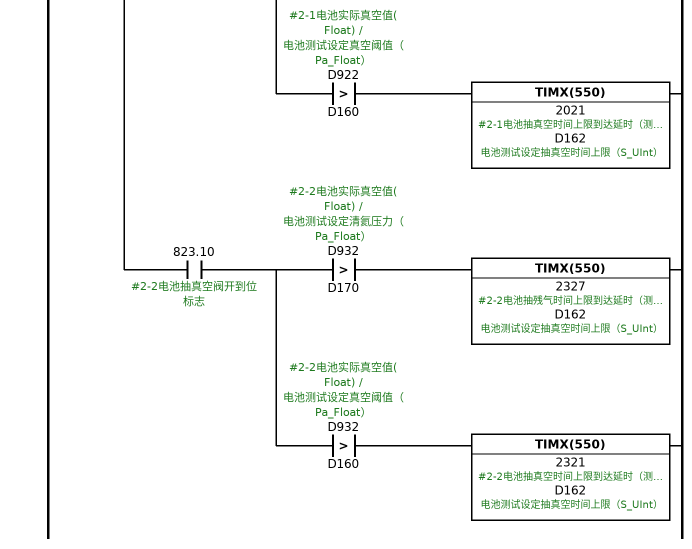
; rung 13
LD P_On
OUT TR0
AND<=F(332) D922 D160  ; #2-1电池实际真空值(Float), 电池测试设定真空阈值（Pa_Float）
LD 823.08  ; #2-1电池抽真空阀开到位标志
OR P_On
ANDLD
TIMX(550) 2020 #1  ; #2-1电池抽真空阈值到达延时（测试）
LD TR0
AND<=F(332) D932 D160  ; #2-2电池实际真空值(Float), 电池测试设定真空阈值（Pa_Float）
LD 823.10  ; #2-2电池抽真空阀开到位标志
OR P_On
ANDLD
TIMX(550) 2320 #1  ; #2-2电池抽真空阈值到达延时（测试）
LD TR0
LD>F(333) D922 D172  ; #2-1电池实际真空值(Float), 电池测试设定破真空阈值（Pa_Float）
OR H5.15  ; 腔体模式（0-正压 1-负压）
ANDLD
TIMX(550) 2022 #1  ; #2-1电池破真空阈值到达延时（测试）
LD TR0
LD>F(333) D932 D172  ; #2-2电池实际真空值(Float), 电池测试设定破真空阈值（Pa_Float）
OR H5.15  ; 腔体模式（0-正压 1-负压）
ANDLD
TIMX(550) 2322 #1  ; #2-2电池破真空阈值到达延时（测试）
LD TR0
AND>=F(334) D922 D176  ; #2-1电池实际真空值(Float), 电池测试设定注氦压力（Pa_Float）
AND 823.12  ; #2-1电池注氦阀开到位标志
TIMHX(551) 2024 #0  ; #2-1电池注氦压力到达延时（测试）
LD TR0
AND>=F(334) D932 D176  ; #2-2电池实际真空值(Float), 电池测试设定注氦压力（Pa_Float）
AND 823.14  ; #2-2电池注氦阀开到位标志
TIMHX(551) 2324 #0  ; #2-2电池注氦压力到达延时（测试）
LD TR0
AND<=F(332) D922 D172  ; #2-1电池实际真空值(Float), 电池测试设定破真空阈值（Pa_Float）
AND 824.00  ; #2-1电池破真空阀开到位标志
TIMX(550) 2023 &20  ; #2-1电池破真空时间上限到达延时（测试）
LD TR0
AND<=F(332) D932 D172  ; #2-2电池实际真空值(Float), 电池测试设定破真空阈值（Pa_Float）
AND 824.02  ; #2-2电池破真空阀开到位标志
TIMX(550) 2323 &20  ; #2-2电池破真空时间上限到达延时（测试）
LD TR0
AND<=F(332) D922 D170  ; #2-1电池实际真空值(Float), 电池测试设定清氦压力（Pa_Float）
TIMX(550) 2026 #1  ; #2-1电池抽残气压力到达延时（测试）
LD TR0
AND<=F(332) D932 D170  ; #2-2电池实际真空值(Float), 电池测试设定清氦压力（Pa_Float）
TIMX(550) 2326 #1  ; #2-2电池抽残气压力到达延时（测试）
LD TR0
AND>=F(334) D922 D174  ; #2-1电池实际真空值(Float), 电池测试设定预抽检测压力（Pa_Float）
AND T2009  ; #2-1腔体预抽时间到达延时（测试）
TIMHX(551) 2028 #0  ; #2-1电池预抽压力正常判定延时（测试）
LD TR0
AND>=F(334) D932 D174  ; #2-2电池实际真空值(Float), 电池测试设定预抽检测压力（Pa_Float）
AND T2009  ; #2-1腔体预抽时间到达延时（测试）
TIMHX(551) 2328 #0  ; #2-2电池预抽压力正常判定延时（测试）
LD TR0
AND 823.12  ; #2-1电池注氦阀开到位标志
AND<F(331) D922 D176  ; #2-1电池实际真空值(Float), 电池测试设定注氦压力（Pa_Float）
TIMX(550) 2025 D168  ; 电池测试设定注氦时间上限（S_UInt）, #2-1电池注氦时间上限到达延时（测试）
LD TR0
AND 823.14  ; #2-2电池注氦阀开到位标志
AND<F(331) D932 D178  ; #2-2电池实际真空值(Float), 注氦压力下限值（Pa_Float）
TIMX(550) 2325 D168  ; 电池测试设定注氦时间上限（S_UInt）, #2-2电池注氦时间上限到达延时（测试）
LD TR0
AND 823.08  ; #2-1电池抽真空阀开到位标志
OUT TR1
AND>F(333) D922 D170  ; #2-1电池实际真空值(Float), 电池测试设定清氦压力（Pa_Float）
TIMX(550) 2027 D162  ; 电池测试设定抽真空时间上限（S_UInt）, #2-1电池抽残气时间上限到达延时（测试）
LD TR1
AND>F(333) D922 D160  ; #2-1电池实际真空值(Float), 电池测试设定真空阈值（Pa_Float）
TIMX(550) 2021 D162  ; 电池测试设定抽真空时间上限（S_UInt）, #2-1电池抽真空时间上限到达延时（测试）
LD TR0
AND 823.10  ; #2-2电池抽真空阀开到位标志
OUT TR0
AND>F(333) D932 D170  ; #2-2电池实际真空值(Float), 电池测试设定清氦压力（Pa_Float）
TIMX(550) 2327 D162  ; 电池测试设定抽真空时间上限（S_UInt）, #2-2电池抽残气时间上限到达延时（测试）
LD TR0
AND>F(333) D932 D160  ; #2-2电池实际真空值(Float), 电池测试设定真空阈值（Pa_Float）
TIMX(550) 2321 D162  ; 电池测试设定抽真空时间上限（S_UInt）, #2-2电池抽真空时间上限到达延时（测试）

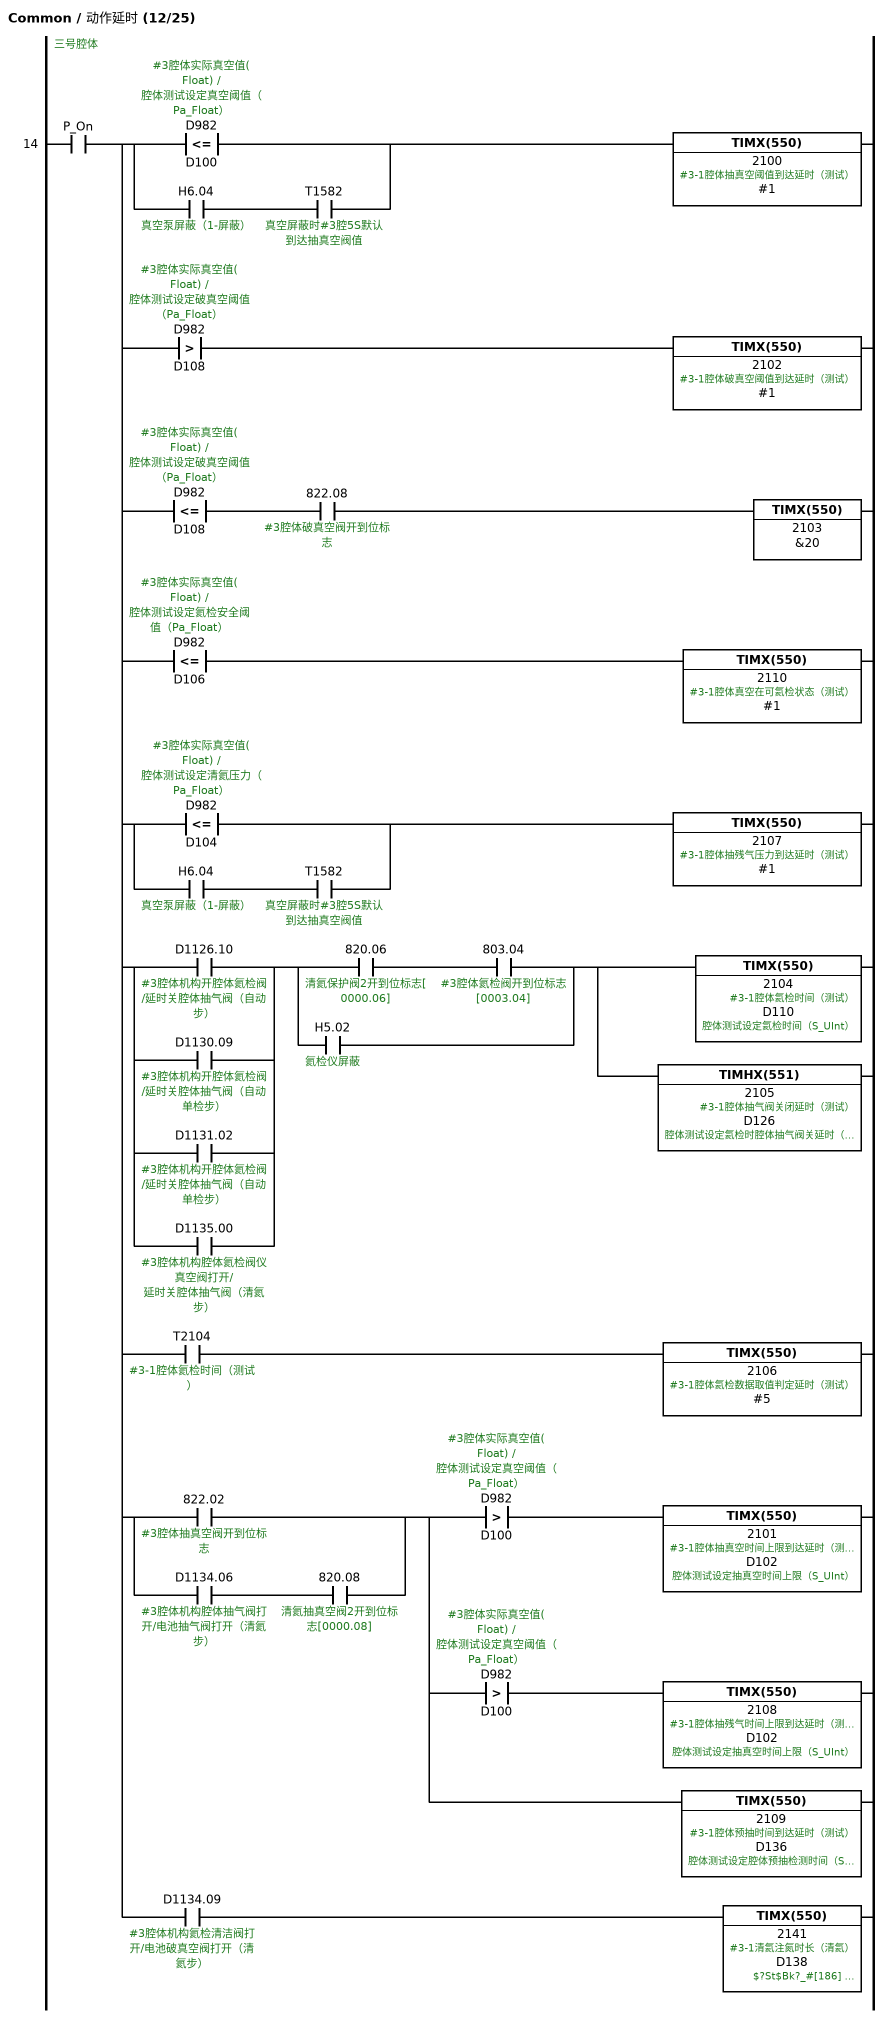
; rung 14: 三号腔体
LD P_On
OUT TR0
LD<=F(332) D982 D100  ; #3腔体实际真空值(Float), 腔体测试设定真空阈值（Pa_Float）
LD H6.04  ; 真空泵屏蔽（1-屏蔽）
AND T1582  ; 真空屏蔽时#3腔5S默认到达抽真空阀值
ORLD
ANDLD
TIMX(550) 2100 #1  ; #3-1腔体抽真空阈值到达延时（测试）
LD TR0
AND>F(333) D982 D108  ; #3腔体实际真空值(Float), 腔体测试设定破真空阈值（Pa_Float）
TIMX(550) 2102 #1  ; #3-1腔体破真空阈值到达延时（测试）
LD TR0
AND<=F(332) D982 D108  ; #3腔体实际真空值(Float), 腔体测试设定破真空阈值（Pa_Float）
AND 822.08  ; #3腔体破真空阀开到位标志
TIMX(550) 2103 &20
LD TR0
AND<=F(332) D982 D106  ; #3腔体实际真空值(Float), 腔体测试设定氦检安全阈值（Pa_Float）
TIMX(550) 2110 #1  ; #3-1腔体真空在可氦检状态（测试）
LD TR0
LD<=F(332) D982 D104  ; #3腔体实际真空值(Float), 腔体测试设定清氦压力（Pa_Float）
LD H6.04  ; 真空泵屏蔽（1-屏蔽）
AND T1582  ; 真空屏蔽时#3腔5S默认到达抽真空阀值
ORLD
ANDLD
TIMX(550) 2107 #1  ; #3-1腔体抽残气压力到达延时（测试）
LD TR0
LD D1126.10  ; #3腔体机构开腔体氦检阀/延时关腔体抽气阀（自动步）
OR D1130.09  ; #3腔体机构开腔体氦检阀/延时关腔体抽气阀（自动单检步）
OR D1131.02  ; #3腔体机构开腔体氦检阀/延时关腔体抽气阀（自动单检步）
OR D1135.00  ; #3腔体机构腔体氦检阀仪真空阀打开/延时关腔体抽气阀（清氦步）
ANDLD
LD 820.06  ; 清氦保护阀2开到位标志[0000.06]
AND 803.04  ; #3腔体氦检阀开到位标志[0003.04]
OR H5.02  ; 氦检仪屏蔽
ANDLD
TIMX(550) 2104 D110  ; 腔体测试设定氦检时间（S_UInt）, #3-1腔体氦检时间（测试）
TIMHX(551) 2105 D126  ; 腔体测试设定氦检时腔体抽气阀关延时（S_UInt）, #3-1腔体抽气阀关闭延时（测试）
LD TR0
AND T2104  ; #3-1腔体氦检时间（测试）
TIMX(550) 2106 #5  ; #3-1腔体氦检数据取值判定延时（测试）
LD TR0
LD 822.02  ; #3腔体抽真空阀开到位标志
LD D1134.06  ; #3腔体机构腔体抽气阀打开/电池抽气阀打开（清氦步）
AND 820.08  ; 清氦抽真空阀2开到位标志[0000.08]
ORLD
ANDLD
OUT TR1
AND>F(333) D982 D100  ; #3腔体实际真空值(Float), 腔体测试设定真空阈值（Pa_Float）
TIMX(550) 2101 D102  ; 腔体测试设定抽真空时间上限（S_UInt）, #3-1腔体抽真空时间上限到达延时（测试）
LD TR1
AND>F(333) D982 D100  ; #3腔体实际真空值(Float), 腔体测试设定真空阈值（Pa_Float）
TIMX(550) 2108 D102  ; 腔体测试设定抽真空时间上限（S_UInt）, #3-1腔体抽残气时间上限到达延时（测试）
LD TR1
TIMX(550) 2109 D136  ; 腔体测试设定腔体预抽检测时间（S_UInt）, #3-1腔体预抽时间到达延时（测试）
LD TR0
AND D1134.09  ; #3腔体机构氦检清洁阀打开/电池破真空阀打开（清氦步）
TIMX(550) 2141 D138  ; $?St$Bk?_#[186] / 管路清氦注氮时间（S_UInt） / $?St$Bk?_#[186], #3-1清氦注氮时长（清氦）

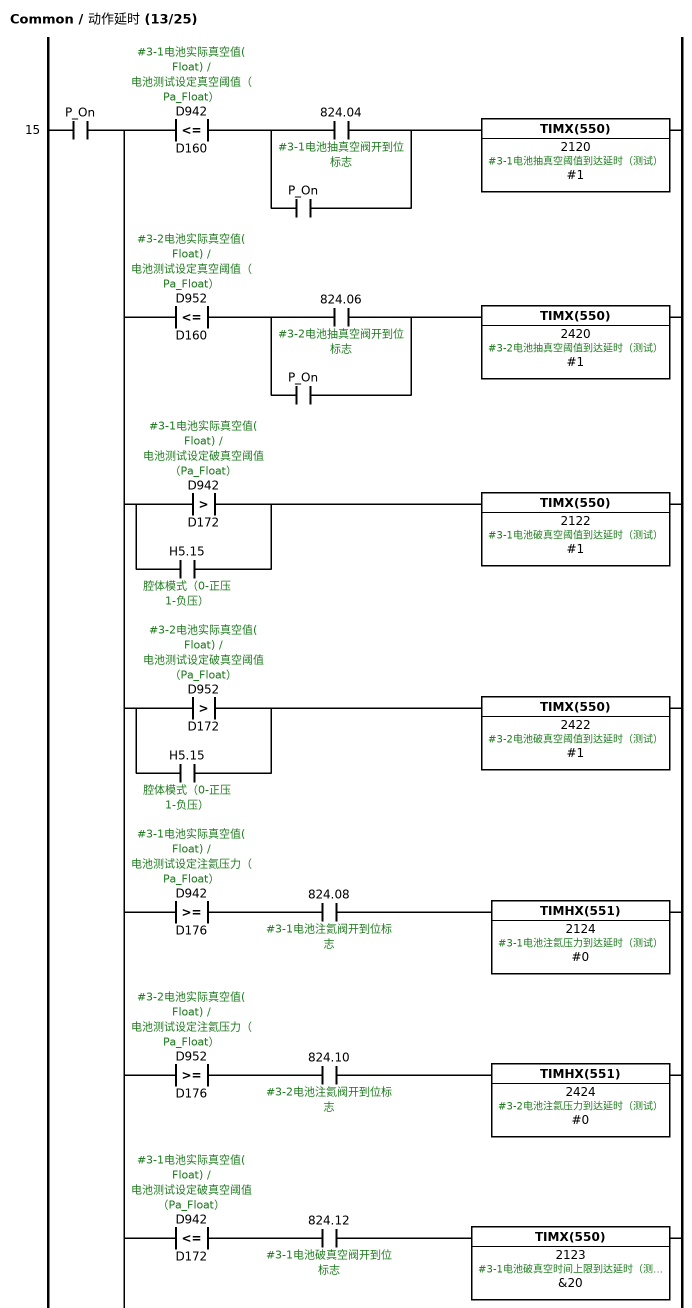

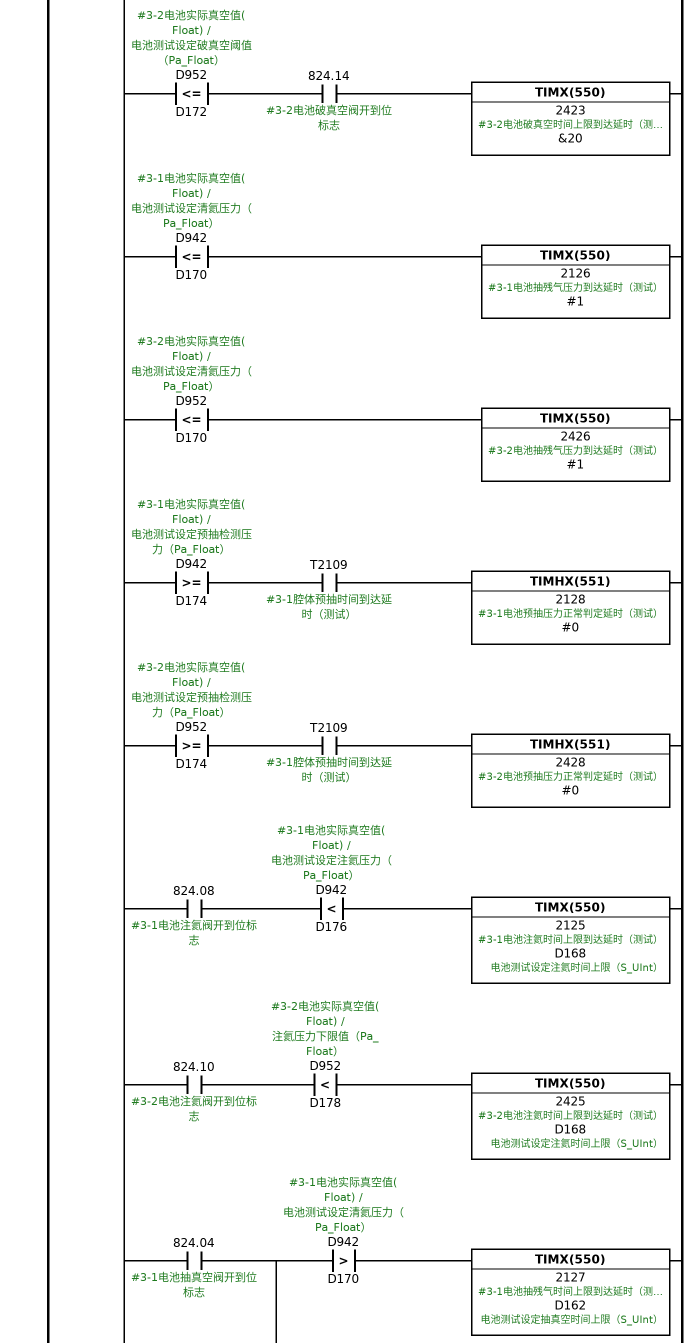

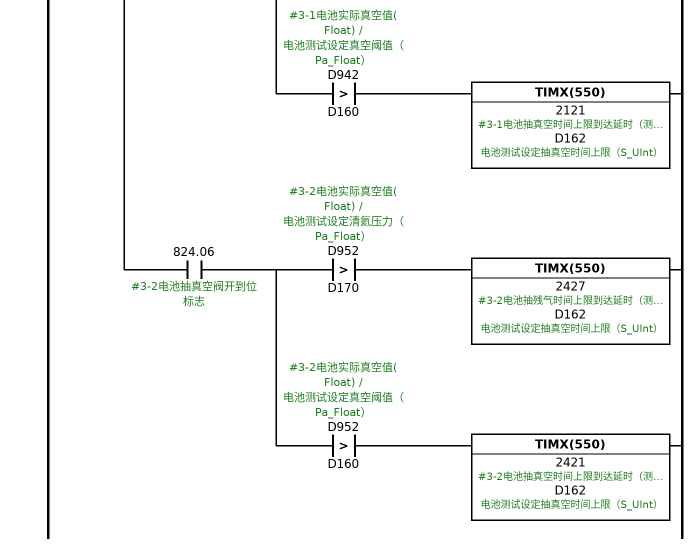
; rung 15
LD P_On
OUT TR0
AND<=F(332) D942 D160  ; #3-1电池实际真空值(Float), 电池测试设定真空阈值（Pa_Float）
LD 824.04  ; #3-1电池抽真空阀开到位标志
OR P_On
ANDLD
TIMX(550) 2120 #1  ; #3-1电池抽真空阈值到达延时（测试）
LD TR0
AND<=F(332) D952 D160  ; #3-2电池实际真空值(Float), 电池测试设定真空阈值（Pa_Float）
LD 824.06  ; #3-2电池抽真空阀开到位标志
OR P_On
ANDLD
TIMX(550) 2420 #1  ; #3-2电池抽真空阈值到达延时（测试）
LD TR0
LD>F(333) D942 D172  ; #3-1电池实际真空值(Float), 电池测试设定破真空阈值（Pa_Float）
OR H5.15  ; 腔体模式（0-正压 1-负压）
ANDLD
TIMX(550) 2122 #1  ; #3-1电池破真空阈值到达延时（测试）
LD TR0
LD>F(333) D952 D172  ; #3-2电池实际真空值(Float), 电池测试设定破真空阈值（Pa_Float）
OR H5.15  ; 腔体模式（0-正压 1-负压）
ANDLD
TIMX(550) 2422 #1  ; #3-2电池破真空阈值到达延时（测试）
LD TR0
AND>=F(334) D942 D176  ; #3-1电池实际真空值(Float), 电池测试设定注氦压力（Pa_Float）
AND 824.08  ; #3-1电池注氦阀开到位标志
TIMHX(551) 2124 #0  ; #3-1电池注氦压力到达延时（测试）
LD TR0
AND>=F(334) D952 D176  ; #3-2电池实际真空值(Float), 电池测试设定注氦压力（Pa_Float）
AND 824.10  ; #3-2电池注氦阀开到位标志
TIMHX(551) 2424 #0  ; #3-2电池注氦压力到达延时（测试）
LD TR0
AND<=F(332) D942 D172  ; #3-1电池实际真空值(Float), 电池测试设定破真空阈值（Pa_Float）
AND 824.12  ; #3-1电池破真空阀开到位标志
TIMX(550) 2123 &20  ; #3-1电池破真空时间上限到达延时（测试）
LD TR0
AND<=F(332) D952 D172  ; #3-2电池实际真空值(Float), 电池测试设定破真空阈值（Pa_Float）
AND 824.14  ; #3-2电池破真空阀开到位标志
TIMX(550) 2423 &20  ; #3-2电池破真空时间上限到达延时（测试）
LD TR0
AND<=F(332) D942 D170  ; #3-1电池实际真空值(Float), 电池测试设定清氦压力（Pa_Float）
TIMX(550) 2126 #1  ; #3-1电池抽残气压力到达延时（测试）
LD TR0
AND<=F(332) D952 D170  ; #3-2电池实际真空值(Float), 电池测试设定清氦压力（Pa_Float）
TIMX(550) 2426 #1  ; #3-2电池抽残气压力到达延时（测试）
LD TR0
AND>=F(334) D942 D174  ; #3-1电池实际真空值(Float), 电池测试设定预抽检测压力（Pa_Float）
AND T2109  ; #3-1腔体预抽时间到达延时（测试）
TIMHX(551) 2128 #0  ; #3-1电池预抽压力正常判定延时（测试）
LD TR0
AND>=F(334) D952 D174  ; #3-2电池实际真空值(Float), 电池测试设定预抽检测压力（Pa_Float）
AND T2109  ; #3-1腔体预抽时间到达延时（测试）
TIMHX(551) 2428 #0  ; #3-2电池预抽压力正常判定延时（测试）
LD TR0
AND 824.08  ; #3-1电池注氦阀开到位标志
AND<F(331) D942 D176  ; #3-1电池实际真空值(Float), 电池测试设定注氦压力（Pa_Float）
TIMX(550) 2125 D168  ; 电池测试设定注氦时间上限（S_UInt）, #3-1电池注氦时间上限到达延时（测试）
LD TR0
AND 824.10  ; #3-2电池注氦阀开到位标志
AND<F(331) D952 D178  ; #3-2电池实际真空值(Float), 注氦压力下限值（Pa_Float）
TIMX(550) 2425 D168  ; 电池测试设定注氦时间上限（S_UInt）, #3-2电池注氦时间上限到达延时（测试）
LD TR0
AND 824.04  ; #3-1电池抽真空阀开到位标志
OUT TR1
AND>F(333) D942 D170  ; #3-1电池实际真空值(Float), 电池测试设定清氦压力（Pa_Float）
TIMX(550) 2127 D162  ; 电池测试设定抽真空时间上限（S_UInt）, #3-1电池抽残气时间上限到达延时（测试）
LD TR1
AND>F(333) D942 D160  ; #3-1电池实际真空值(Float), 电池测试设定真空阈值（Pa_Float）
TIMX(550) 2121 D162  ; 电池测试设定抽真空时间上限（S_UInt）, #3-1电池抽真空时间上限到达延时（测试）
LD TR0
AND 824.06  ; #3-2电池抽真空阀开到位标志
OUT TR0
AND>F(333) D952 D170  ; #3-2电池实际真空值(Float), 电池测试设定清氦压力（Pa_Float）
TIMX(550) 2427 D162  ; 电池测试设定抽真空时间上限（S_UInt）, #3-2电池抽残气时间上限到达延时（测试）
LD TR0
AND>F(333) D952 D160  ; #3-2电池实际真空值(Float), 电池测试设定真空阈值（Pa_Float）
TIMX(550) 2421 D162  ; 电池测试设定抽真空时间上限（S_UInt）, #3-2电池抽真空时间上限到达延时（测试）

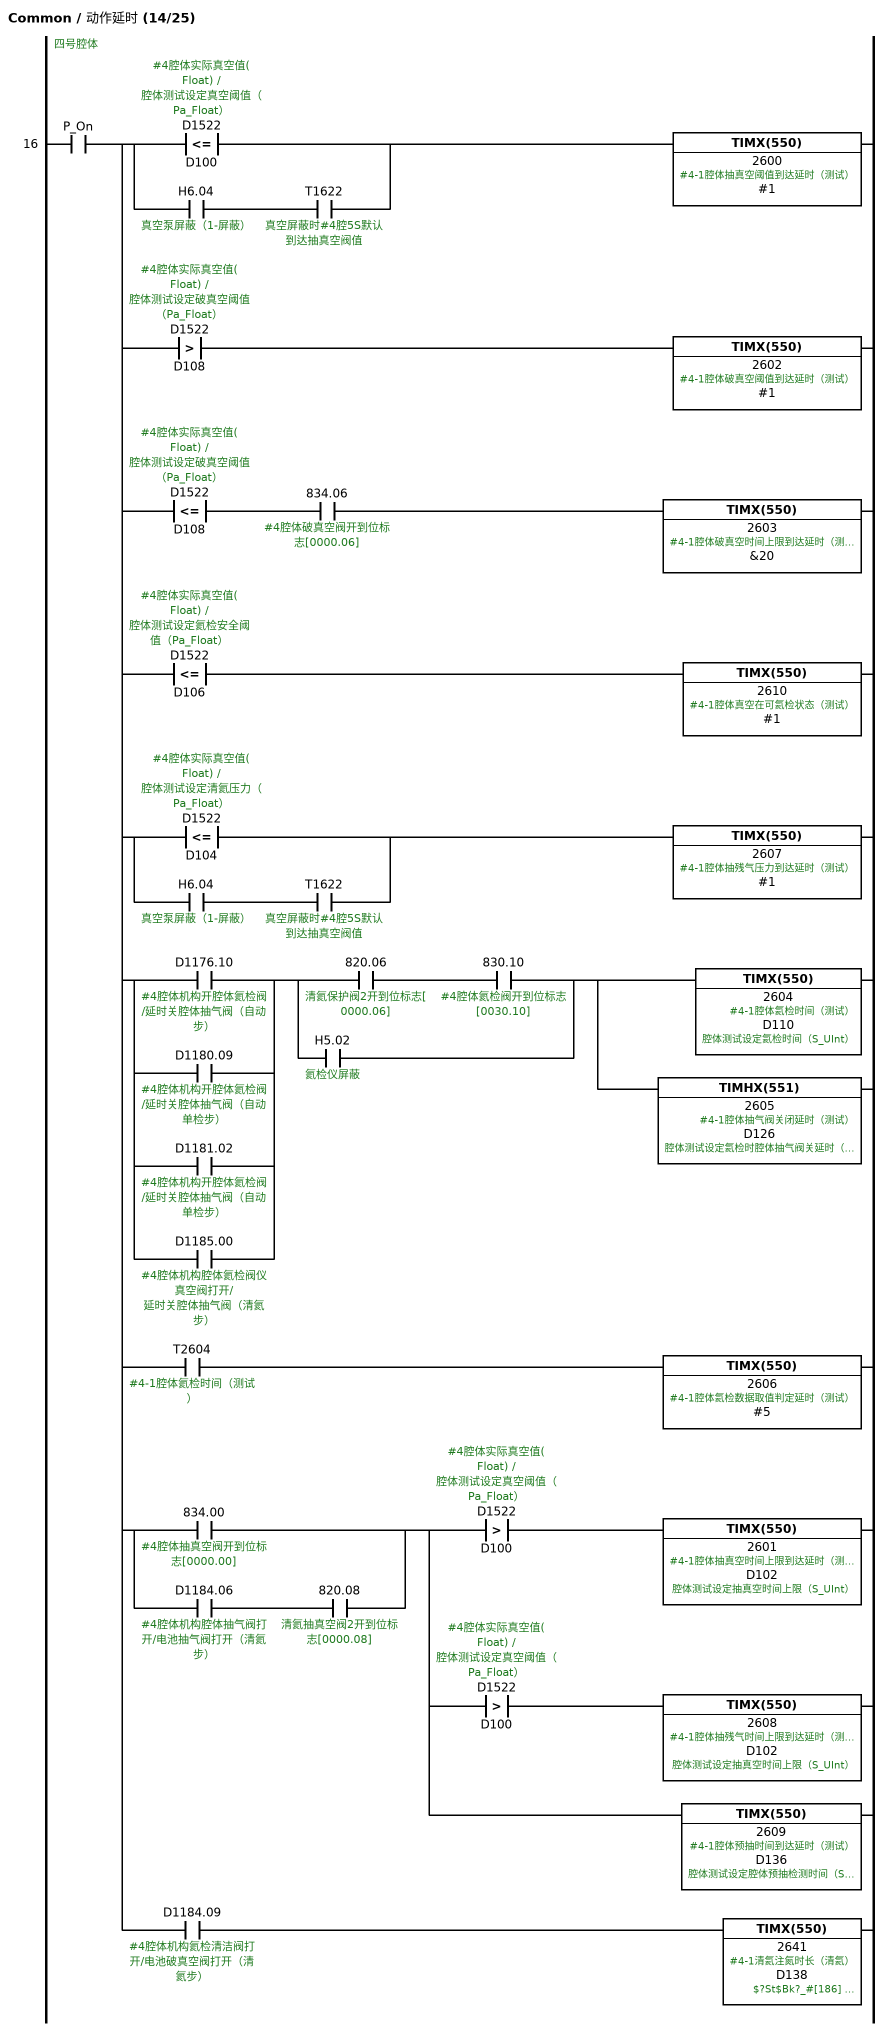
; rung 16: 四号腔体
LD P_On
OUT TR0
LD<=F(332) D1522 D100  ; #4腔体实际真空值(Float), 腔体测试设定真空阈值（Pa_Float）
LD H6.04  ; 真空泵屏蔽（1-屏蔽）
AND T1622  ; 真空屏蔽时#4腔5S默认到达抽真空阀值
ORLD
ANDLD
TIMX(550) 2600 #1  ; #4-1腔体抽真空阈值到达延时（测试）
LD TR0
AND>F(333) D1522 D108  ; #4腔体实际真空值(Float), 腔体测试设定破真空阈值（Pa_Float）
TIMX(550) 2602 #1  ; #4-1腔体破真空阈值到达延时（测试）
LD TR0
AND<=F(332) D1522 D108  ; #4腔体实际真空值(Float), 腔体测试设定破真空阈值（Pa_Float）
AND 834.06  ; #4腔体破真空阀开到位标志[0000.06]
TIMX(550) 2603 &20  ; #4-1腔体破真空时间上限到达延时（测试）
LD TR0
AND<=F(332) D1522 D106  ; #4腔体实际真空值(Float), 腔体测试设定氦检安全阈值（Pa_Float）
TIMX(550) 2610 #1  ; #4-1腔体真空在可氦检状态（测试）
LD TR0
LD<=F(332) D1522 D104  ; #4腔体实际真空值(Float), 腔体测试设定清氦压力（Pa_Float）
LD H6.04  ; 真空泵屏蔽（1-屏蔽）
AND T1622  ; 真空屏蔽时#4腔5S默认到达抽真空阀值
ORLD
ANDLD
TIMX(550) 2607 #1  ; #4-1腔体抽残气压力到达延时（测试）
LD TR0
LD D1176.10  ; #4腔体机构开腔体氦检阀/延时关腔体抽气阀（自动步）
OR D1180.09  ; #4腔体机构开腔体氦检阀/延时关腔体抽气阀（自动单检步）
OR D1181.02  ; #4腔体机构开腔体氦检阀/延时关腔体抽气阀（自动单检步）
OR D1185.00  ; #4腔体机构腔体氦检阀仪真空阀打开/延时关腔体抽气阀（清氦步）
ANDLD
LD 820.06  ; 清氦保护阀2开到位标志[0000.06]
AND 830.10  ; #4腔体氦检阀开到位标志[0030.10]
OR H5.02  ; 氦检仪屏蔽
ANDLD
TIMX(550) 2604 D110  ; 腔体测试设定氦检时间（S_UInt）, #4-1腔体氦检时间（测试）
TIMHX(551) 2605 D126  ; 腔体测试设定氦检时腔体抽气阀关延时（S_UInt）, #4-1腔体抽气阀关闭延时（测试）
LD TR0
AND T2604  ; #4-1腔体氦检时间（测试）
TIMX(550) 2606 #5  ; #4-1腔体氦检数据取值判定延时（测试）
LD TR0
LD 834.00  ; #4腔体抽真空阀开到位标志[0000.00]
LD D1184.06  ; #4腔体机构腔体抽气阀打开/电池抽气阀打开（清氦步）
AND 820.08  ; 清氦抽真空阀2开到位标志[0000.08]
ORLD
ANDLD
OUT TR1
AND>F(333) D1522 D100  ; #4腔体实际真空值(Float), 腔体测试设定真空阈值（Pa_Float）
TIMX(550) 2601 D102  ; 腔体测试设定抽真空时间上限（S_UInt）, #4-1腔体抽真空时间上限到达延时（测试）
LD TR1
AND>F(333) D1522 D100  ; #4腔体实际真空值(Float), 腔体测试设定真空阈值（Pa_Float）
TIMX(550) 2608 D102  ; 腔体测试设定抽真空时间上限（S_UInt）, #4-1腔体抽残气时间上限到达延时（测试）
LD TR1
TIMX(550) 2609 D136  ; 腔体测试设定腔体预抽检测时间（S_UInt）, #4-1腔体预抽时间到达延时（测试）
LD TR0
AND D1184.09  ; #4腔体机构氦检清洁阀打开/电池破真空阀打开（清氦步）
TIMX(550) 2641 D138  ; $?St$Bk?_#[186] / 管路清氦注氮时间（S_UInt） / $?St$Bk?_#[186], #4-1清氦注氮时长（清氦）

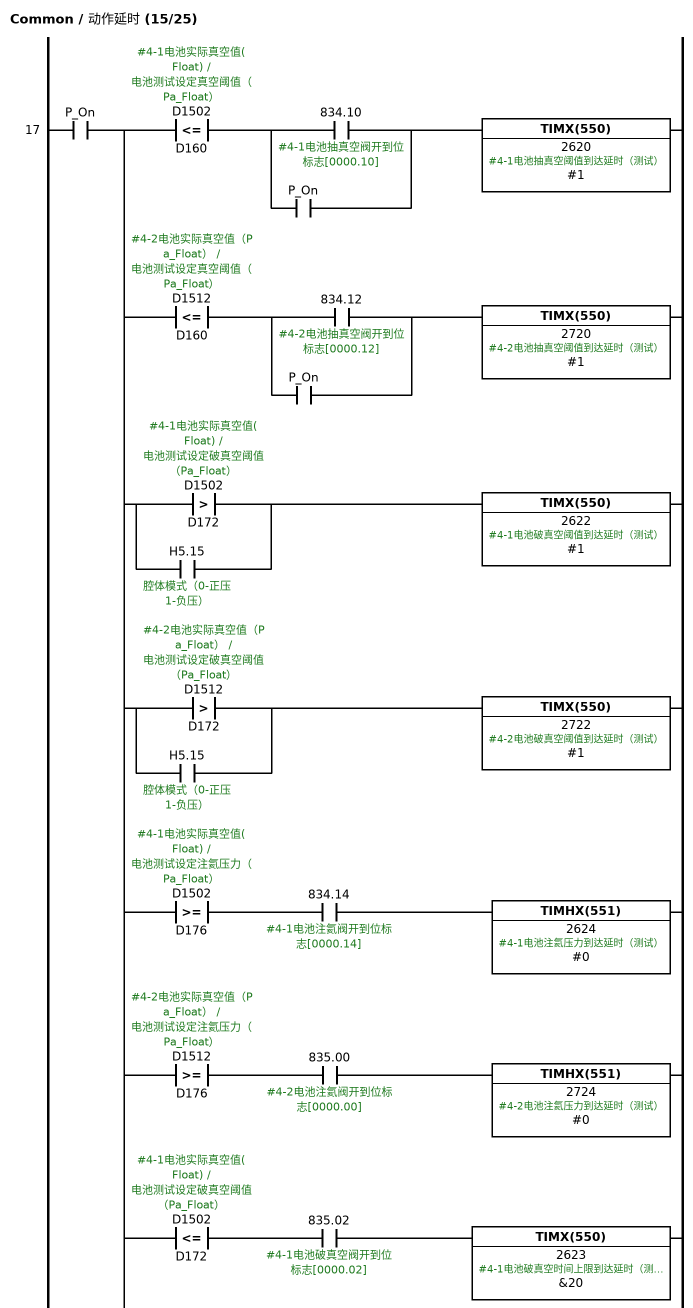

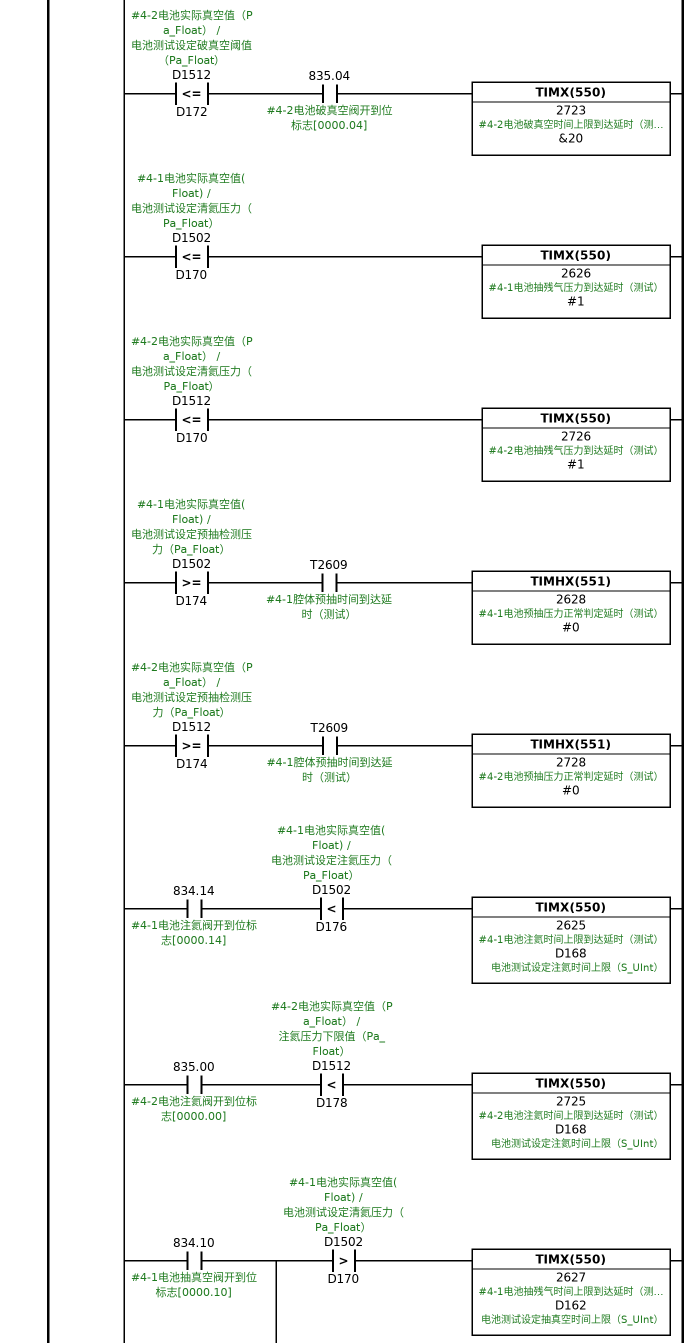

